# B&R Automation Studio project TD52 (part 118)

#### OUT_HACyclic.st - Cyclic code
```iecst
(*******************************************************************************
AGGR: copy OUT PVs for module HalIO (cyclic)

This code is confidential and proprietary to the INNIO Company.
It may not be used in any form, or reproduced in any manner, without the express
written permission of the INNIO Company.
Copyright, INNIO Company, 2022

Customized modifications: -
------------------------

History:
-------
V3.99	14-06-2012	Weitzer, generated FOR modular software
V4.00	14-02-2014	Weitzer, change version number
V4.00.1	29.10.2014	Weitzer, set Pact to 0 if GCB is open and -10kW < P < 10kW
V4.03	11-02-2015	Weitzer, add OUT_HA.szEng_Motorversion
		20-04-2015	Weitzer, add MORIS safety loop to MM2VIS structure
		16-09-2015	Weitzer, add MM2VIS.rP_ActUnfilt[1] for hi-res trending
		21-09-2015	Weitzer, add rI_MaxL1..3 to OUT_HA for monitoring
V4.04	17-01-2017	Denk, add IPC status OUT variables
V4.04.1	23-02-2017	Weitzer, correct current dynamic calculation
V4.05	12-09-2017	Denk, add OUT_HA.bSimWinMOD_withoutBus_Active
		27-07-2017	Messner, CAN Diagnosis Variables added
		20-12-2017	Weitzer, change bus bar voltages to standard IO format
		21-01-2018	Perktold,hardware operation mode switch added
		12.02.2018	lettenb. MM2VIS.rF_MMD_BusBar[] added
V4.05.1 14-02-2018	Weitzer, change TJ overview CAN diag. data to FAST comm.
V4.05.2 19-03-2018	Denk, WinMOD simulation ON/OFF logic added
V4.07.0	24-01-2019	Schmid, MM2VIS for MMD serial number added
V4.08	18-07-2019	Denk, IPC status logic changed because of new PPC3100 (new OUT_HA.iT_CFast2)
V4.11.0	18-03-2022	Perktold, tiTimeout von 2s auf 5s erhöht (erhöhte DGS Stabilität)
V4.12	28-10-2022	Weitzer, added auto detect multiplier for bus bar and synch voltages > 30kV
V4.14	19-11-2024	Farre,	 added auto detect multiplier for grid voltage (2024-236)

Instructions for use:
--------------------
-

Outstandings:
------------
*******************************************************************************)

PROGRAM _CYCLIC

	(* Visu out *)
	FOR ucCount := 1 TO 2 DO

		(* OUT VISU *)
		MM2VIS.rI_L1[ucCount] 			:= tI_L1[ucCount].Ai; 					(* current 1 *)
		MM2VIS.rI_L2[ucCount]			:= tI_L2[ucCount].Ai; 					(* current 2 *)
		MM2VIS.rI_L3[ucCount] 			:= tI_L3[ucCount].Ai; 					(* current 3 *)
		MM2VIS.rI_Dyn[ucCount]	 		:= UINT_TO_REAL(usIDyn[ucCount])/1000; 	(* current dynamic *)
		IF Para.rI_GenNom[ucCount] <> 0 THEN
			MM2VIS.rI_Dyn[ucCount] := UINT_TO_REAL(usIDyn[ucCount])/Para.rI_GenNom[ucCount]; 	(* current dynamic *)
		END_IF;
		MM2VIS.rI_N[ucCount] 			:= INT_TO_REAL(ssIN[ucCount]); 			(* current neutral *)
		IF ssSynchAngleDeviation[ucCount] > 1800 THEN 	(* angle deviation synchronization  +180° - -180° *)
			MM2VIS.rAng_MMD_Diff[ucCount] 	:= INT_TO_REAL(ssSynchAngleDeviation[ucCount]-3600)/10;
		ELSE
			MM2VIS.rAng_MMD_Diff[ucCount] 	:= INT_TO_REAL(ssSynchAngleDeviation[ucCount])/10;
		END_IF;

		(* visualisation of synchronization mode *)
		IF bSyncSlipMode[ucCount] THEN
			MM2VIS.iIdx_MMD_SynchMode[ucCount] := 1;
		ELSIF bSyncCheckMode[ucCount] THEN
			MM2VIS.iIdx_MMD_SynchMode[ucCount] := 2;
		ELSIF bSyncDeadBusMode[ucCount] THEN
			MM2VIS.iIdx_MMD_SynchMode[ucCount] := 3;
		ELSE
			MM2VIS.iIdx_MMD_SynchMode[ucCount] := 0;
		END_IF;

		MM2VIS.rMMD_HW_Version[ucCount]	:= UINT_TO_REAL(usMMDSynchHWVariant[ucCount])/100;			(* program version MMD *)
		MM2VIS.rU_MMD_Diff[ucCount] 	:= INT_TO_REAL(ssSynchVoltDeviation[ucCount]) * rMul_MMD_U_Synch[ucCount]; 		(* votage deviation synchronization *)
		sMMD_SerialNumber				:= UDINT_TO_STRING(ulMMDSerialNumber[ucCount]);
		MM2VIS.sMMD_SerialNumber[ucCount]	:= REPLACE(	IN1:= '00000000000', 						(* SerialNumber MMD *)
														IN2:= sMMD_SerialNumber,
														L:= LEN(sMMD_SerialNumber), P:= 11 - LEN(sMMD_SerialNumber) + 1);
		iMMD_ModuleID					:= usMMDModuleID[ucCount];
		IF iMMD_ModuleID <= 9999 THEN
			sMMD_ModuleID := UINT_TO_STRING(iMMD_ModuleID);
			sMMD_ModuleID := REPLACE(IN1:= '0000', IN2:= sMMD_ModuleID, L:= LEN(sMMD_ModuleID), P:= 4 - LEN(sMMD_ModuleID) + 1);
			MM2VIS.sMMD_SerialNumber[ucCount] := REPLACE(	IN1:= MM2VIS.sMMD_SerialNumber[ucCount], 				(* ModuleID MMD *)
															IN2:= sMMD_ModuleID,
															L:= 4, P:= 1);
		ELSE
			sMMD_ModuleID := '0000';
			FOR iIdx_ModuleID := 3 TO 0 BY -1 DO
				iMMD_ModuleID_Char	:= TRUNC(UINT_TO_REAL(iMMD_ModuleID)/16**iIdx_ModuleID);
				CASE iMMD_ModuleID_Char OF
					15:		sMMD_ModuleID	:= REPLACE(IN1:= sMMD_ModuleID, IN2:= 'F', L:= 1, P:= (4 - iIdx_ModuleID));
					14:		sMMD_ModuleID	:= REPLACE(IN1:= sMMD_ModuleID, IN2:= 'E', L:= 1, P:= (4 - iIdx_ModuleID));
					13:		sMMD_ModuleID	:= REPLACE(IN1:= sMMD_ModuleID, IN2:= 'D', L:= 1, P:= (4 - iIdx_ModuleID));
					12:		sMMD_ModuleID	:= REPLACE(IN1:= sMMD_ModuleID, IN2:= 'C', L:= 1, P:= (4 - iIdx_ModuleID));
					11:		sMMD_ModuleID	:= REPLACE(IN1:= sMMD_ModuleID, IN2:= 'B', L:= 1, P:= (4 - iIdx_ModuleID));
					10:		sMMD_ModuleID	:= REPLACE(IN1:= sMMD_ModuleID, IN2:= 'A', L:= 1, P:= (4 - iIdx_ModuleID));
					ELSE	sMMD_Temp		:= INT_TO_STRING(iMMD_ModuleID_Char);
							sMMD_ModuleID	:= REPLACE(IN1:= sMMD_ModuleID, IN2:= sMMD_Temp, L:= 1, P:= (4 - iIdx_ModuleID));
				END_CASE;
				iMMD_ModuleID		:= iMMD_ModuleID MOD REAL_TO_UINT(16**iIdx_ModuleID);
			END_FOR;
			MM2VIS.sMMD_SerialNumber[ucCount] := REPLACE(IN1:= MM2VIS.sMMD_SerialNumber[ucCount], IN2:= sMMD_ModuleID, L:= 4, P:= 1);
		END_IF;

		MM2VIS.rU_Bus_L1_2[ucCount] 	:= tU_Bus_L1_2[ucCount].Ai * rMul_MMD_U_Bus[ucCount]; 		(* bus bar voltage 1 2 *)
		MM2VIS.rU_Bus_L2_3[ucCount] 	:= tU_Bus_L2_3[ucCount].Ai * rMul_MMD_U_Bus[ucCount]; 		(* bus bar voltage 2 3 *)
		MM2VIS.rU_Bus_L3_1[ucCount] 	:= tU_Bus_L3_1[ucCount].Ai * rMul_MMD_U_Bus[ucCount]; 		(* bus bar voltage 3 1 *)
		MM2VIS.rU_Bus_L1N[ucCount] 		:= tU_Bus_L1N[ucCount].Ai  * rMul_MMD_U_Bus[ucCount]; 		(* bus bar voltage 1 *)
		MM2VIS.rU_Bus_L2N[ucCount] 		:= tU_Bus_L2N[ucCount].Ai  * rMul_MMD_U_Bus[ucCount]; 		(* bus bar voltage 2 *)
		MM2VIS.rU_Bus_L3N[ucCount] 		:= tU_Bus_L3N[ucCount].Ai  * rMul_MMD_U_Bus[ucCount]; 		(* bus bar voltage 3 *)

		(* OUT HAL_IO VIS *)
		MM2VIS.rPF_Act[ucCount]			:= tPF_Act[ucCount].Ai; 									(* power factor *)
		MM2VIS.rI_Avg[ucCount] 			:= tI_Avg[ucCount].Ai;										(* current average *)
		MM2VIS.rP_Act[ucCount]			:= tP_Act[ucCount].Ai * rMul_MMD_U_Gen[ucCount]; 			(*  actual electric power [kW] *)
		MM2VIS.rP_ActUnfilt[ucCount]	:= tP_Act[ucCount].Unfilt * rMul_MMD_U_Gen[ucCount];		(*  actual unfiltered electric power [kW] *)
		(* set to 0 kW when generator switch is open *)
		IF NOT tGCB_On.Di THEN
			IF (MM2VIS.rP_Act[1] > -10) AND (MM2VIS.rP_Act[1] < 10) THEN	(* and actual power within +/- 10 kW *)
				MM2VIS.rP_Act[1]       := 0;
				MM2VIS.rP_ActUnfilt[1] := 0;
	 		END_IF;
		END_IF;

		MM2VIS.rQ_Act[ucCount]			:= tQ_Act[ucCount].Ai 		 * rMul_MMD_U_Gen[ucCount];		(* reactive power [kVar] *)
		MM2VIS.rS_Act[ucCount]			:= tS_Act[ucCount].Ai 		 * rMul_MMD_U_Gen[ucCount];		(* power apperent *)
		MM2VIS.rU_MMD_Synch1[ucCount] 	:= tU_MMD_Synch1[ucCount].Ai * rMul_MMD_U_Synch[ucCount];	(* synchronization voltage 1 *)
		MM2VIS.rU_MMD_Synch2[ucCount] 	:= tU_MMD_Synch2[ucCount].Ai * rMul_MMD_U_Synch[ucCount];	(* synchronization voltage 2 *)
		MM2VIS.rU_Avg[ucCount] 			:= tU_Avg[ucCount].Ai 		 * rMul_MMD_U_Gen[ucCount];		(* voltage average *)
		MM2VIS.rU_L1N[ucCount]			:= tU_L1N[ucCount].Ai 		 * rMul_MMD_U_Gen[ucCount];		(* voltage 1 *)
		MM2VIS.rU_L1L2[ucCount]			:= tU_L1L2[ucCount].Ai 		 * rMul_MMD_U_Gen[ucCount];		(* voltage 12 *)
		MM2VIS.rU_L2N[ucCount]			:= tU_L2N[ucCount].Ai 		 * rMul_MMD_U_Gen[ucCount];		(* voltage 2 *)
		MM2VIS.rU_L2L3[ucCount]			:= tU_L2L3[ucCount].Ai 		 * rMul_MMD_U_Gen[ucCount];		(* voltage 23 *)
		MM2VIS.rU_L3N[ucCount]			:= tU_L3N[ucCount].Ai 		 * rMul_MMD_U_Gen[ucCount];		(* voltage 3 *)
		MM2VIS.rU_L3L1[ucCount]			:= tU_L3L1[ucCount].Ai 		 * rMul_MMD_U_Gen[ucCount]; 	(* voltage 31 *)
		MM2VIS.rF_MMD[ucCount] 			:= tF_MMD[ucCount].Ai;										(* frequency multi measure device *)
		MM2VIS.rF_MMD_Synch1[ucCount] 	:= tF_MMD_Synch1[ucCount].Ai; 								(* Frequency Sync-network 1 *)
		MM2VIS.rF_MMD_Synch2[ucCount] 	:= tF_MMD_Synch2[ucCount].Ai; 								(* Frequency Sync-network 2 *)
		MM2VIS.rF_MMD_BusBar[ucCount] 	:= tF_MMD_BusBar[ucCount].Ai; 								(* frequency bus bar *)
		MM2VIS.rMMD_FW_Version[ucCount]	:= DINT_TO_REAL(tMMD_FW_Version[ucCount].Ai)/100;			(*program version MMD firmware*)

		(* feedback synch DO *)
		TOF_SyImp[ucCount](IN := bMMD_SynchDO[ucCount],PT := T#2s);
		MM2VIS.bMMD_SynchDO[ucCount] := TOF_SyImp[ucCount].Q;

		(* U diff bar graphs MAX value (limit times 2) *)
		MM2VIS.rUDiffMaxScale[ucCount] := Para.rU_DiffMax[ucCount] * Para.rU_SyncNom[ucCount] * 2;

		(* f diff bar graphs MIN and MAX value (limit times 2) *)
		MM2VIS.rF_DiffMaxScale[ucCount] := Para.rF_DiffMax[ucCount] * 2;
		MM2VIS.rF_DiffMinScale[ucCount] := Para.rF_DiffMin[ucCount] * 2;

		(* copy maximum current values to out structure *)
		OUT_HA.rI_MaxL1[ucCount] := MM2VIS.rI_MaxL1[ucCount];
		OUT_HA.rI_MaxL2[ucCount] := MM2VIS.rI_MaxL2[ucCount];
		OUT_HA.rI_MaxL3[ucCount] := MM2VIS.rI_MaxL3[ucCount];

	END_FOR;

	(* Status MORIS safety loop for visualization *)
	MM2VIS.bMO_SaftyLoop := tMO_SaftyLoop.Di;

	(* gasmixer stepper card B&R X20 SM1426 *)
	OUT_HA.iGM1_MStepActPos; 	(*gasmixer 1 - Actual position from SM1426-Module [Microsteps]*)	(*OldName: slGM1_MStepActPos_TC1; Cycle: 5;*)
	OUT_HA.iGM1_Status;			(*gasmixer 1 - Status Word from SM1426-Module*)						(*OldName: usGM1_Status_TC1; Cycle: 5;*)
	OUT_HA.iGM2_MStepActPos;	(*gasmixer 2 - Actual position from SM1426-Module [Microsteps]*)	(*OldName: slGM2_MStepActPos_TC1; Cycle: 5;*)
	OUT_HA.iGM2_Status;			(*gasmixer 2 - Status Word from SM1426-Module*)						(*OldName: usGM2_Status_TC1; Cycle: 5;*)

	(* Copy motor version string to out structure *)
	OUT_HA.szEng_Motorversion := Para.szEng_Motorversion;

	(* Copy order ID string to out structure *)
	OUT_HA.szOrderID := Para.szOrderID;

	(* Copy order ID string to out structure *)
	OUT_HA.iEngID := VIS2MM.iEngID;

	(* IPC status *)

	OUT_HA.iSerialNumber_CPU;	(*Serial number CPU*)
	OUT_HA.iModulID_CPU;		(*Modul ID CPU*)
	OUT_HA.iPowerOnCycles;		(*Power On cycles CPU*)
	OUT_HA.iOperatingHours_CPU; (*Operating hours CPU*)
	OUT_HA.iBatterieStatus; 	(*Batterie Status IPC*)
	OUT_HA.iT_CPU; 				(*Temperature CPU*)
	OUT_HA.iT_CPU_PLC; 			(*Temperature PLC X20CP368xX CPU*)
	OUT_HA.iT_Board; 			(*Temperature Board*)
	OUT_HA.iT_Chipset;			(*Temperature Chipset*)
	OUT_HA.iT_PS; 				(*Temperature IPC board power supply*)
	OUT_HA.iT_CFast; 			(*Temperature IPC CFast*)
	OUT_HA.iT_CFast2; 			(*Temperature IPC CFast2*)

	(* WinMOD simulation for IPC status *)
	IF OUT_HA.bSimWinMOD_Active THEN
		OUT_HA.iBatterieStatus := TRUE;
	END_IF;

	(* WinMOD simulation with/without bus hardware *)
	OUT_HA.bSimWinMOD_withoutBus_Active; 	(* TRUE = without bus hardware *)

	(* WinMOD simulation ON/OFF *)
	xTON_WatchdogSIM2AR0(IN:= NOT bWatchdogSIM2AR, PT:= tiTimeout);
	xTON_WatchdogSIM2AR1(IN:= bWatchdogSIM2AR, PT:= tiTimeout);
	IF (xTON_WatchdogSIM2AR0.Q OR xTON_WatchdogSIM2AR1.Q) THEN
		OUT_HA.bSimWinMOD_Active := FALSE;
	ELSE
		OUT_HA.bSimWinMOD_Active := TRUE;
	END_IF;

	(* Status CAN BUS for Visualization *)
	MM2VIS.iCANopen_CMS_status 	:= CANopen_CMS.status;
	MM2VIS.iCANopen_CMS_info 	:= CANopen_CMS.info;
	MM2VIS.iCMSmain_Init_status	:= MAX(CMSmain_Init.status, CMSmain_Init2.status);

	(* Status CAN IC900 all Modules for Visualization *)
	MM2VIS.iIC900_AllErrEventMax 	:= IN_HA.iE_IgnStat;
	MM2VIS.iIC900_AllErrCount 		:= IN_HA.iIC900CommErrCount;
	MM2VIS.iIC900_AllErrMax 		:= ucIC900CommErrMax;
	MM2VIS.iIC900_AllPhaseCnt 		:= usIC900PhaseCnt;
	MM2VIS.iIC900_AllErrAvg			:= usIC900CommErrAvg;

	(* Status CAN Monic all Modules for Visualization *)
	MM2VIS.iMonic_AllErrEventMax 	:= IN_HA.iEMonStatus;
	MM2VIS.iMonic_AllErrCount 		:= IN_HA.iMonicCommErrCount;
	MM2VIS.iMonic_AllErrMax 		:= ucMonicCommErrMax;
	MM2VIS.iMonic_AllPhaseCnt 		:= usMonicPhaseCnt;
	MM2VIS.iMonic_AllErrAvg			:= usMonicCommErrAvg;

	(* Status CAN TecJet all Modules for Visualization - SLOW monitoring not needed *)
//	MM2VIS.iTecJet_AllErrEventMax 	:= ucTecJetCommErrEventMax;
//	MM2VIS.iTecJet_AllErrCount 		:= IN_HA.iTecJetCommErrCount;
//	MM2VIS.iTecJet_AllErrSlowMax 	:= ucTecJetCommErrSlowMax;
//	MM2VIS.iTecJet_AllSlowPhaseCnt 	:= usTecJetSlowPhaseCnt;
//	MM2VIS.iTecJet_AllErrSlowAvg	:= usTecJetCommErrSlowAvg;

	(* Status CAN TecJet individual Modules for Visualization *)
	MM2VIS.iTecJet_AllErrEventMax 	:= 0;
	MM2VIS.iTecJet_AllErrCount 		:= 0;
	MM2VIS.iTecJet_AllErrSlowMax 	:= 0;
	MM2VIS.iTecJet_AllSlowPhaseCnt 	:= 0;
	MM2VIS.iTecJet_AllErrSlowAvg	:= 0;
	FOR ucLoopCnt := 1 TO 4 DO
		MM2VIS.iTecJet_ErrEventMax[ucLoopCnt] 	:= IN_HA.tE_TEC[ucLoopCnt].Contr[0];
		MM2VIS.iTecJet_ErrMaxCur[ucLoopCnt]		:= IN_HA.iTecErrCnt[ucLoopCnt];
		MM2VIS.iTecJet_ErrMax[ucLoopCnt] 		:= usTecJetCommErrFastMax[ucLoopCnt];
		MM2VIS.iTecJet_PhaseCnt[ucLoopCnt] 		:= usTecJetFastPhaseCnt[ucLoopCnt];
		MM2VIS.iTecJet_ErrAvgCnt[ucLoopCnt] 	:= usTecJetCommErrFastAvg[ucLoopCnt];

		MM2VIS.iTecJet_AllErrEventMax 	:= MAX(MM2VIS.iTecJet_AllErrEventMax , MM2VIS.iTecJet_ErrEventMax[ucLoopCnt]);
		MM2VIS.iTecJet_AllErrCount 		:= MAX(MM2VIS.iTecJet_AllErrCount    , MM2VIS.iTecJet_ErrMaxCur[ucLoopCnt]);
		MM2VIS.iTecJet_AllErrSlowMax 	:= MAX(MM2VIS.iTecJet_AllErrSlowMax  , MM2VIS.iTecJet_ErrMax[ucLoopCnt]);
		MM2VIS.iTecJet_AllSlowPhaseCnt 	:= MAX(MM2VIS.iTecJet_AllSlowPhaseCnt, MM2VIS.iTecJet_PhaseCnt[ucLoopCnt]);
		MM2VIS.iTecJet_AllErrSlowAvg	:= MAX(MM2VIS.iTecJet_AllErrSlowAvg  , MM2VIS.iTecJet_ErrAvgCnt[ucLoopCnt]);
	END_FOR;

	(* Status CAN KLS98 all Modules for Visualization *)
	MM2VIS.iKLS98_AllErrEventMax 	:= ucKLS98CommErrEventMax;
	MM2VIS.iKLS98_AllErrMaxCur 		:= ucKLS98CommErrMaxCur;
	MM2VIS.iKLS98_AllErrMax 		:= ucKLS98CommErrMaxAll;
	MM2VIS.iKLS98_AllPhaseCntMax 	:= usKLS98PhaseCntMax;
	MM2VIS.iKLS98_AllErrAvgMax		:= usKLS98CommErrAvgMax;

	(* Status CAN KLS98 individual Modules for Visualization *)
	FOR ucLoopCnt := 1 TO xEngType.NumberOfCylinder DO
		MM2VIS.iKLS98_ErrEventMax[ucLoopCnt] 	:= IN_HA.tE_KLS[ucLoopCnt].conf[99];
		MM2VIS.iKLS98_ErrMaxCur[ucLoopCnt]		:= IN_HA.iKLS98CommErrCount[ucLoopCnt];
		MM2VIS.iKLS98_ErrMax[ucLoopCnt] 		:= ucKLS98CommErrMax[ucLoopCnt];
		MM2VIS.iKLS98_PhaseCnt[ucLoopCnt] 		:= usKLS98PhaseCnt[ucLoopCnt];
		MM2VIS.iKLS98_ErrAvgCnt[ucLoopCnt] 		:= usKLS98CommErrAvg[ucLoopCnt];
	END_FOR;

	(* Status CAN SAFI all Modules for Visualization *)
	MM2VIS.iSAFI_AllErrEventMax := ucSAFICommErrEventMax;
	MM2VIS.iSAFI_AllErrMaxCur 	:= usSAFICommErrMaxCur;
	MM2VIS.iSAFI_AllErrMax		:= usSAFICommErrMaxAll;
	MM2VIS.iSAFI_AllPhaseCntMax	:= usSAFIPhaseCntMax;
	MM2VIS.iSAFI_AllErrAvgMax	:= usSAFICommErrAvgMaxCnt;

	(* Status CAN SAFI individual Modules for Visualization *)
	FOR ucLoopCnt := 1 TO xEngType.NumberOfCylinder/2 DO
		MM2VIS.iSAFI_ErrEventMax[ucLoopCnt] := IN_HA.tE_SAFI[ucLoopCnt].sdata[1];
		MM2VIS.iSAFI_ErrMaxCur[ucLoopCnt]	:= IN_HA.iCnt_SA_ComErr[ucLoopCnt] / 100;
		MM2VIS.iSAFI_ErrMax[ucLoopCnt] 		:= usSAFICommErrMax[ucLoopCnt];
		MM2VIS.iSAFI_PhaseCnt[ucLoopCnt] 	:= usSAFIPhaseCnt[ucLoopCnt];
		MM2VIS.iSAFI_ErrAvgCnt[ucLoopCnt] 	:= usSAFICommErrAvgCnt[ucLoopCnt];
	END_FOR;

	(* H A R D W A R E   S W I T C H E S *)
	(* GoodQual for HMI *)
	OUT_HA.tHW_Switches.bGoodQual	:=  tDI_OMS_Man.GoodQual AND tDI_OMS_Auto.GoodQual AND tDI_RMS_On.GoodQual AND tDI_RMS_Remote.GoodQual AND tDI_SyOMS_Man.GoodQual AND tDI_SyOMS_Auto.GoodQual;
	(* Hardware operation mode switch *)
	xTON_OMS.IN := NOT tDI_OMS_Man.Di AND NOT tDI_OMS_Auto.Di;
	xTON_OMS();
	IF NOT tDI_OMS_Man.Di AND NOT tDI_OMS_Auto.Di AND xTON_OMS.Q THEN
		OUT_HA.tHW_Switches.iIdx_OMS_Hw 	:= 0;
	ELSIF tDI_OMS_Man.Di AND NOT tDI_OMS_Auto.Di THEN
		OUT_HA.tHW_Switches.iIdx_OMS_Hw 	:= 1;
	ELSIF NOT tDI_OMS_Man.Di AND tDI_OMS_Auto.Di THEN
		OUT_HA.tHW_Switches.iIdx_OMS_Hw 	:= 2;
	END_IF;

	(* Hardware request mode switch *)
	xTON_RMS.IN := NOT tDI_RMS_On.Di AND NOT tDI_RMS_Remote.Di;
	xTON_RMS();
	IF NOT tDI_RMS_On.Di AND NOT tDI_RMS_Remote.Di AND xTON_RMS.Q THEN
		OUT_HA.tHW_Switches.iIdx_RMS_Hw 	:= 0;
	ELSIF tDI_RMS_On.Di AND NOT tDI_RMS_Remote.Di THEN
		OUT_HA.tHW_Switches.iIdx_RMS_Hw 	:= 1;
	ELSIF NOT tDI_RMS_On.Di AND tDI_RMS_Remote.Di THEN
		OUT_HA.tHW_Switches.iIdx_RMS_Hw 	:= 2;
	END_IF;

	(* Hardware synchronisation operation mode switch *)
	xTON_SyOMS.IN := NOT tDI_SyOMS_Man.Di AND NOT tDI_SyOMS_Auto.Di;
	xTON_SyOMS();
	IF NOT tDI_SyOMS_Man.Di AND NOT tDI_SyOMS_Auto.Di AND xTON_SyOMS.Q THEN
		OUT_HA.tHW_Switches.iIdx_SyOMS_Hw 	:= 0;
	ELSIF tDI_SyOMS_Man.Di AND NOT tDI_SyOMS_Auto.Di THEN
		OUT_HA.tHW_Switches.iIdx_SyOMS_Hw 	:= 1;
	ELSIF NOT tDI_SyOMS_Man.Di AND tDI_SyOMS_Auto.Di THEN
		OUT_HA.tHW_Switches.iIdx_SyOMS_Hw 	:= 2;
	END_IF;

	(* MMU Information for custom module (bus applications) *)
	OUT_HA.rI_Dyn 				:=	MM2VIS.rI_Dyn;
	OUT_HA.rI_GenUnbalanced 	:=	MM2VIS.rI_GenUnbalanced;
	OUT_HA.rU_MMD_Diff 			:=	MM2VIS.rU_MMD_Diff;
	OUT_HA.iIdx_MMD_SynchMode 	:=	MM2VIS.iIdx_MMD_SynchMode;

END_PROGRAM
```

#### OUT_HAInit.st - Init code
```iecst
(*******************************************************************************
AGGR: copy OUT PVs for module HalIO (init)

This code is confidential and proprietary to the INNIO Company.
It may not be used in any form, or reproduced in any manner, without the express
written permission of the INNIO Company.
Copyright, INNIO Company, 2019

Customized modifications: -
------------------------

History:
-------
V3.99	06-03-2013	Weitzer, generated FOR modular software
V4.00	14-02-2014	Weitzer, change version number
V4.05	21-01-2018	Perktold,hardware operation mode switch added
V4.07	15-05-2019	Zengerer Init call for detection of missing tHA2GR items in init

Instructions for use:
--------------------
-

Outstandings:
------------
*******************************************************************************)

PROGRAM _INIT

	(* call to get a addresses for the HalIO Fub of OUT HAL_IO VIS variables *)

	PF_Act; 			(* power factor *)
	I_Avg;				(* current average *)
	P_Act; 				(*  actual electric power [kW] *)
	Q_Act; 				(* reactive power [kVar] *)
	S_Act; 				(* power apperent *)
	U_MMD_Synch1; 		(* synchronization voltage 1 *)
	U_MMD_Synch2; 		(* synchronization voltage 2 *)
	U_Avg; 				(* voltage average *)
	U_L1N; 				(* voltage 1 *)
	U_L1L2;				(* voltage 12 *)
	U_L2N; 				(* voltage 2 *)
	U_L2L3; 			(* voltage 23 *)
	U_L3N; 				(* voltage 3 *)
	U_L3L1;				(* voltage 31 *)
	F_MMD;				(* frequency multi measure device *)
	F_MMD_Synch1; 		(* Frequency Sync-network 1 *)
	F_MMD_Synch2; 		(* Frequency Sync-network 2 *)
	MMD_FW_Version;		(*program version MMD firmware*)

	xTON_OMS.PT		:= T#1s; 	(* Delaytime for changing position of HW-switch *)
	xTON_RMS.PT 	:= T#1s;	(* Delaytime for changing position of HW-switch *)
	xTON_SyOMS.PT 	:= T#1s;	(* Delaytime for changing position of HW-switch *)

	(*Init call for detection of missing tHA2GR items *)
	tHA2GR.bCheck_HA2GR ;
	tHA2GR.tU_Droop.GoodQual ;

	tHA2CU.tSet_U_Droop_COn.GoodQual ;

END_PROGRAM
```

#### OUT_HA.var - Local variables
```iecst
(********************************************************************
 * COPYRIGHT -- INNIO Company
 ********************************************************************
 * Program: IN_HA
 * File: IN_HA.var
 * Author: weitzert
 * Created: June 14, 2012
 ********************************************************************
 * Local variables of program IN_HA
 ********************************************************************)
VAR
	ucCount : USINT;
	TOF_SyImp : ARRAY[0..2] OF TOF;
	xTON_OMS : TON;
	xTON_RMS : TON;
	xTON_SyOMS : TON;
	tiTimeout : TIME := T#5s;
	xTON_WatchdogSIM2AR0 : TON;
	xTON_WatchdogSIM2AR1 : TON;
	sMMD_SerialNumber : STRING[11];
	iMMD_ModuleID : UINT;
	iMMD_ModuleID_Char : INT;
	iIdx_ModuleID : INT;
	sMMD_ModuleID : STRING[4];
	sMMD_Temp : STRING[1];
END_VAR
```

### Program Logical/HalIO/MsgHA (IEC, version 4.11.0) - + HalIO Messages

- MsgHACyclic.st (not readable text: treated as protected, skipped)

- MsgHAInit.st (not readable text: treated as protected, skipped)

#### MsgHA.var
```iecst
VAR
	iCount : USINT := 0;
	iAdrAmmBase2MM : UDINT;
	iAdrMM2AmmBase : UDINT;
	xMsg3311 : Msg;
	xMsg2399 : Msg;
	xMsg2400 : Msg;
	xMsg9400 : Msg;
	xMsg9386 : Msg; (*Plant Communication configuration failed*)
	xMsg9384 : Msg; (*Plant Communication Interrupted*)
	xMsg9391 : Msg; (*Plant Communication force active*)
END_VAR
```

### Program Logical/HalIO/ParHA (IEC, version 4.07.0) - + HalIO Parameter

- perm_par.st (not readable text: treated as protected, skipped)

#### perm_par.var
```iecst
VAR
	tParaIntern : ParaHandler_typ; (*Connector type to perm_par*)
	tMM2ParaBase_ReadBack : MM2ParaBase_type; (*INTERNAL! V4.06 new readback structure for information from previous tasks*)
	bWriteDataObj : BOOL; (* TRUE=write data object module *)
	bDataObjLenErr : BOOL; (*Error occured in permem: data module size missmatch*)
	bCreateDataObj : BOOL; (* TRUE=create new data object *)
	bWriteOnce : BOOL; (* write permanent memory once *)
	DatObjCreate_01 : DatObjCreate; (* data object create *)
	DatObjInfoBak_02 : DatObjInfo; (* data object info *)
	DatObjDelete_01 : DatObjDelete; (* data object delete *)
	DatObjRead_01 : DatObjRead; (* data object read *)
	DatObjRead_02 : DatObjRead; (* manual initiated data object read *)
	DatObjWrite_01 : DatObjWrite; (* data object write *)
	DatObjDelete_02 : DatObjDelete; (* data object delete *)
	DatObjDelete_11 : DatObjDelete; (*Delete Backup File*)
	DatObjInfo_01 : DatObjInfo; (* data object info *)
	DatObjInfo_02 : DatObjInfo; (* data object info *)
	szModuleName : STRING[35]; (* module name of object *)
	szModuleNameBackup : STRING[35]; (* module name of posiibly created backup object *)
	DatObjCopy_01 : DatObjCopy;
	bCopyDataObj : BOOL;
	TON_WarnDelay : TON;
	TON_WritePMEM : TON; (* delay write permanent memory *)
	ulPMPointer : UDINT; (* adress of actual checksum value *)
	ulChecksum : UDINT; (* parameter checksum value *)
	pm_len : UDINT; (* permanent value lenght *)
	ulChecksumOld : UDINT; (* last vlaue of parameter checksum *)
	ulChkValue : UDINT; (* actual value of parameter pointer *)
	pm_id : UDINT; (* permanent value identifier *)
	pm_p : UDINT; (* permanent value pointer *)
	DatObjInfo_META : DatObjInfo;
	DatObjRead_META : DatObjRead;
	szMetaDataRaw : STRING[2000];
	szMetaData : ARRAY[0..4] OF STRING[35];
	szMetaDataVis : ARRAY[0..3] OF STRING[35];
	ssIndex : INT;
	ssCount : INT;
	ucMetaDataRaw : ARRAY[0..2000] OF USINT;
	ssCount2 : INT;
	szMetaDataFile : STRING[10];
	szText1 : STRING[20];
	pv_adr_IN_XX_tPB2MM : UDINT;
	pv_lng : UDINT;
	pv_lng_IN_XX_tPB2MM : UDINT;
	pv_lng_OUT_XX_tPB2MM : UDINT;
	szText2 : STRING[20];
	pv_adr_OUT_XX_tXX2PB : UDINT;
END_VAR
VAR CONSTANT
	ERR_NOERROR : UINT := 0;
END_VAR
VAR
	usPMWriteCnt : UINT;
	pm_Error : UDINT; (* permanent value error *) (* Deleted: pm : ParaMem_typ; permanent memory tags mathias, 22.8.11*)
	fun_Error : UDINT := 0; (*state > 0 = function error*)
	xLocalParaCheck : ParaCheckFUB; (*local function instance to check parameter values*)
	TON_ParaSetupOk : TON;
	bParaCheckSystemOk : BOOL;
	iDebug_ParaOkChecked : UDINT;
	bRestoreBackupDataObj : BOOL := FALSE;
	bRestoreDataObjContent : BOOL := FALSE;
	pm_id_backup : UDINT;
	pm_p_Backup : UDINT;
	DatObjCopy_02 : DatObjCopy;
	bDeleteBackupDataObj : BOOL := FALSE; (*Command to delete backup data module file on purpose*)
	bDebugPara : ARRAY[0..5] OF BOOL;
	ssIndex2 : INT;
	ssIndex3 : INT;
	ssIndex4 : INT;
	ssIndexVis : INT;
	szText : STRING[40];
	pv_adr_Para : UDINT;
	szParaSnippet : ARRAY[0..5] OF STRING[150];
	szParaIndex : STRING[10];
	slValue : DINT;
	iModuleDLD_ResetCount : INT;
	bDownloadDetected : BOOL;
	bFlagParaStructCopyWorking : BOOL; (*true, if cyclic para copying is active, 1 false cycle at every copy *)
	bStoreInitParaInDataObj : BOOL := FALSE;
	bTestflag : BOOL;
	bReadOutMETA_Once : BOOL;
	tParaCheck_iPvAdress : ARRAY[0..5] OF UDINT;
	tParaCheck_iPvLengt : ARRAY[0..5] OF UDINT;
	tParaCheck_rPvValue : ARRAY[0..5] OF REAL;
	tParaCheck_rRangeMIN : ARRAY[0..5] OF REAL;
	tParaCheck_rRangeMAX : ARRAY[0..5] OF REAL;
	tParaCheck_szPvName : ARRAY[0..5] OF STRING[35];
	ssFormatDetected : INT;
	szMetaDataPart : STRING[150];
	szFullTaskName : STRING[35];
	szFullMetaModuleName : STRING[35];
	debugLen : INT;
	debugSize : INT := 0;
	strcat_adr1 : UDINT;
	strcat_adr2 : UDINT;
	ssIndexTN : INT;
	bAlternate : BOOL;
	n : INT;
	iAlternateChecksum : DINT;
	iAlternateChecksumOld : DINT;
	ulDebugChkValue : ARRAY[0..999] OF UDINT;
	Adr1 : UDINT;
	Adr2 : UDINT;
	usPMWriteCntStepsize : UINT := 1; (*different step sizes to help debug*)
	usPMWriteCntXOR : UINT;
	usPMWriteCntAltSum : UINT;
	ulAdrPM : UDINT;
	usChkValuePM : USINT;
	ulAdrPara : UDINT;
	ulPara_len : UDINT;
	usChkValuePara : USINT;
	iDebugCountPMDifferences : DINT := 0;
	bEngineRunDetected : BOOL; (*detection status bit autocommand 100 /101  for engine run state*)
	ucMetaDataDebugInfoLine : ARRAY[0..24] OF STRING[80];
	ssIndexMand : INT := 0;
	szMetaDataMand : STRING[35];
	iMyErrorInfo_Autoreset : DINT; (*internal autoreset counter*)
	ssIndex_Version : INT; (*internal*)
	ssIndex_BU : INT; (*internal*)
	ssIndex_BU2 : INT; (*internal*)
END_VAR
```

### Package Logical/HalIO/CAN - CAN

### CAN_HA.var
```iecst
(********************************************************************
 * COPYRIGHT -- INNIO Company
 ********************************************************************
 * Package: HAL_IO
 * File: CAN_HA.var
 * Author: Schmid
 * Created: December 7, 2021
 ********************************************************************
 * Variables of package HAL_IO/CAN
 ********************************************************************)
VAR CONSTANT
	iMAX_NUMB_OF_CANMODS : UINT := 20; (*Max. number of CAN modules*)
	iIdxCAN_IGN : UINT := 1; (* Ignition, Tecjet *)
	iIdxCAN_NOxS_IF1 : UINT := 2; (* NOx sensor interface 1 *)
	iIdxCAN_NOxS_IF2 : UINT := 3; (* NOx sensor interface 2 *)
	iIdxCAN_NOxS_IF3 : UINT := 7; (* NOx sensor interface 3 *)
	iIdxCAN_CB : UINT := 4; (* Conrod bearing *)
	iIdxCAN_OQS : UINT := 5; (* Oil quality sensor *)
	iIdxCAN_IGN2 : UINT := 6; (*2nd Ignition CAN line*)
	sCAN_IGN2_ident : STRING[10] := 'IGN2'; (*CAN ID string Ignition 2*)
	sCAN_IGN_ident : STRING[10] := 'IGN1'; (*CAN ID string Ignition 1*)
	sCAN_NOxS_IF1_ident : STRING[10] := 'NOX1'; (*CAN ID string NOx sensor IF1*)
	sCAN_NOxS_IF2_ident : STRING[10] := 'NOX2'; (*CAN ID string NOx sensor IF2*)
	sCAN_NOxS_IF3_ident : STRING[10] := 'NOX3'; (*CAN ID string NOx sensor IF3*)
	sCAN_CB_ident : STRING[10] := 'CRB'; (*CAN ID string Conrod bearing*)
	sCAN_OQS_ident : STRING[10] := 'OQS'; (*CAN ID string oil quality sensor*)
END_VAR
VAR
	xDiagCreateInfo_CAN : DiagCreateInfo; (*Get number of configured modules*)
	xDiagGetStrInfo_CAN : DiagGetStrInfo; (*Get name of configured modules*)
	xDiagDisposeInfo_CAN : DiagDisposeInfo; (*Free ressources of AsIODiag*)
	sLabelInfo : STRING[50]; (*Includes label of configured module*)
	sAddrInfo : STRING[50]; (*Includes address of configured modul*)
	iModPos : ARRAY[0..iMAX_NUMB_OF_CANMODS] OF UDINT; (*Array includes index of used CAN IF cards*)
	iIndex : UDINT; (*Index of actual read module*)
	iIdent : UDINT; (*Ident from xDiagCreateInfo_CAN*)
	iNrEntries : UDINT; (*Number of configured modules from xDiagCreateInfo_CAN*)
	sModSlotSel : ARRAY[0..iMAX_NUMB_OF_CANMODS] OF STRING[50]; (*Slot ID of selected configured CAN modules*)
	sCANAddr : STRING[50]; (*CAN IF PLC address string*)
	iIdxCAN_IF : ARRAY[1..2] OF UINT; (*Index array to assign CAN IF card to according role*)
	iPosCAN : ARRAY[1..2] OF UINT; (*Index array to determine CAN ID string order (for X20CS2770)*)
	iIdxPosCAN : UINT; (*Running index of found CAN IF cards*)
	xTON_CANbusoff : TON; (*CAN bus off timer*)
	xTON_SysRun : TON; (*Timer starting at PLC start*)
END_VAR
```

### Program Logical/HalIO/CAN/caninitHA (IEC, version 4.14.0) - HalIO CAN communication init

#### caninitHACyclic.st
```iecst
(*******************************************************************************
AGGR: intiate CAN communication (cyclic)

This code is confidential and proprietary to the INNIO Company.
It may not be used in any form, or reproduced in any manner, without the express
written permission of the INNIO Company.
Copyright, INNIO Company, 2024

Customized modifications: -
------------------------

History:
-------
V0.1	31-08-2001	Fahringer,	generated from caninit.c V0.2
		31-08-2001	Fahringer,	last modification
V0.21	14-10-2003	Weitzer,	transfer all CAN and CMS FUBs to caninit task
V0.40	14-02-2007  Weitzer,	change to new standard IF (SL1.SS1.IF2)
								delete MMD (multimeasure device)
V0.50	07-09-2007	Weitzer		SAFI added
								main FUB´s moved to canmain program
V0.60	23-02-2010	Weitzer,	SAFI2 (prot injection) added
V3.99.0	07-05-2012	Weitzer		generated for modular software
V4.00	14-02-2014	Weitzer,	change version number
V4.10	03-11-2020	Schmid,		engine CAN node position on node P10 as option (Aggreko standard)
V4.11	07-12-2021	Schmid,		flexible CAN interface detection
		22-12-2021	Andre,		avoid potential array index overrun
V4.12	23-02-2023	Weitzer,	add IGN2 CAN interface
V4.22	18-10-2023	Perktold,	added X20CP368xX CAN interfaces
V4.13	17-10-2023	Andre,		Only perform ARwin warm start if the CAN bus off state cannot be quit
V4.14	28-10-2024	Kafka,		SAFI / KLS21 devices of bank B use 2nd card and the rest use 1st one

Instructions for use:
--------------------
-initiate the CAN-Bus communictation controller
-initiate CAN CMS manager

Outstandings:
------------
*******************************************************************************)

PROGRAM _CYCLIC

	(* Dsiplay hardware path of CAN interface _IF1 *)

	IF MM2VIS.iCAN_HW_Slot = 0 AND IN_HA.tPB2MM.bParaSetupOk THEN

		IF LEFT(sModSlotSel[iIdxCAN_IGN],3) = LEFT(MM2VIS.sCAN_HW_Slot_X20CP368xX,3) THEN
			IF xEngType.Type9 THEN	(* B&R X20CP368xX J920 *)
				MM2VIS.iCAN_HW_Slot :=	9;
				strcpy(ADR(MM2VIS.sCAN_HW_Slot_X20CP368xX_J920), ADR(sModSlotSel[iIdxCAN_IGN]));
			ELSE					(* B&R X20CP368xX *)
				MM2VIS.iCAN_HW_Slot :=	8;
				strcpy(ADR(MM2VIS.sCAN_HW_Slot_X20CP368xX), ADR(sModSlotSel[iIdxCAN_IGN]));
			END_IF;

		ELSIF LEFT(sModSlotSel[iIdxCAN_IGN],3) = LEFT(MM2VIS.sCAN_HW_Slot_IPC_3100,3) THEN
			IF xEngType.Type9 THEN	(* B&R PPC3100 J920 *)
				MM2VIS.iCAN_HW_Slot :=	7;
				strcpy(ADR(MM2VIS.sCAN_HW_Slot_IPC_3100_J920), ADR(sModSlotSel[iIdxCAN_IGN]));
			ELSE					(* B&R PPC3100 *)
				MM2VIS.iCAN_HW_Slot :=	6;
				strcpy(ADR(MM2VIS.sCAN_HW_Slot_IPC_3100), ADR(sModSlotSel[iIdxCAN_IGN]));
			END_IF;

		ELSIF	LEFT(sModSlotSel[iIdxCAN_IGN],3) = LEFT(MM2VIS.sCAN_HW_Slot_IPC,3) THEN
			IF xEngType.Type9 THEN	(* B&R PPC900 J920 *)
				MM2VIS.iCAN_HW_Slot :=	4;
				strcpy(ADR(MM2VIS.sCAN_HW_Slot_IPC_J920), ADR(sModSlotSel[iIdxCAN_IGN]));
			ELSE					(* B&R PPC900 *)
				MM2VIS.iCAN_HW_Slot :=	1;
				strcpy(ADR(MM2VIS.sCAN_HW_Slot_IPC), ADR(sModSlotSel[iIdxCAN_IGN]));
			END_IF;

		ELSIF	LEFT(sModSlotSel[iIdxCAN_IGN],3) = LEFT(MM2VIS.sCAN_HW_Slot_IPC_GE_IP,3) THEN
			IF xEngType.Type9 THEN	(* GE IPC J920 *)
				MM2VIS.iCAN_HW_Slot :=	5;
				strcpy(ADR(MM2VIS.sCAN_HW_Slot_IPC_GE_IP_J920), ADR(sModSlotSel[iIdxCAN_IGN]));
			ELSE					(* GE IPC *)
				MM2VIS.iCAN_HW_Slot :=	3;
				strcpy(ADR(MM2VIS.sCAN_HW_Slot_IPC_GE_IP), ADR(sModSlotSel[iIdxCAN_IGN]));
			END_IF;

		ELSIF	LEFT(sModSlotSel[iIdxCAN_IGN],3) = LEFT(MM2VIS.sCAN_HW_Slot_IPC_CMaU,3) THEN
			(* B&R IPC CM&U *)
			MM2VIS.iCAN_HW_Slot	:=	2;
			strcpy(ADR(MM2VIS.sCAN_HW_Slot_IPC_CMaU), ADR(sModSlotSel[iIdxCAN_IGN]));

		ELSIF LEN(sModSlotSel[iIdxCAN_IGN]) > 0 THEN
			(* default: B&R PPC3100 *)
			MM2VIS.iCAN_HW_Slot :=	6;
			strcpy(ADR(MM2VIS.sCAN_HW_Slot_IPC_3100),	ADR(sModSlotSel[iIdxCAN_IGN]));
		END_IF;

	END_IF;

	(* cyclic call of CAN devices  *)

	IF CMSinit_Init.cms_ident <> 0 THEN		(* check if CMS init was successful *)

		IF IN_HA.tICxx_CanGo.ECANDevGo <> 0 THEN
			IF CANDevGo_InBuffer[IN_HA.tICxx_CanGo.CANDevGo[1]].ECANDevGo = 0 THEN
				CANDevGo_InBuffer[IN_HA.tICxx_CanGo.CANDevGo[1]] := IN_HA.tICxx_CanGo;
			END_IF;
		END_IF;

		IF IN_HA.tMonic_CanGo.ECANDevGo <> 0 THEN
			IF CANDevGo_InBuffer[IN_HA.tMonic_CanGo.CANDevGo[1]].ECANDevGo = 0 THEN
				CANDevGo_InBuffer[IN_HA.tMonic_CanGo.CANDevGo[1]] := IN_HA.tMonic_CanGo;
			END_IF;
		END_IF;

		IF IN_HA.tSAFI_CanGo.ECANDevGo <> 0 THEN
			IF CANDevGo_InBuffer[IN_HA.tSAFI_CanGo.CANDevGo[1]].ECANDevGo = 0 THEN
				CANDevGo_InBuffer[IN_HA.tSAFI_CanGo.CANDevGo[1]] := IN_HA.tSAFI_CanGo;
			END_IF;
		END_IF;

		IF IN_HA.tKLS98_CanGo.ECANDevGo <> 0 THEN
			IF CANDevGo_InBuffer[IN_HA.tKLS98_CanGo.CANDevGo[1]].ECANDevGo = 0 THEN
				CANDevGo_InBuffer[IN_HA.tKLS98_CanGo.CANDevGo[1]] := IN_HA.tKLS98_CanGo;
			END_IF;
		END_IF;

//		Not used at the moment
//		IF IN_HA.tGasMeteringUnit_CanGo.ECANDevGo <> 0 THEN
//			CANDevGo_InBuffer[IN_HA.tGasMeteringUnit_CanGo.CANDevGo[1]] := IN_HA.tGasMeteringUnit_CanGo;
//		END_IF;

		FOR ucDevSequencer := 1 TO 32 DO

			IF CANDevGo_InBuffer[ucDevSequencer].ECANDevGo = 128 THEN
				CANDevGo_InBuffer[ucDevSequencer].ECANDevGo := 0;
				IF ucDevSequencer < 32 THEN
					ucDevSequencer := ucDevSequencer + 1;
				END_IF;
			END_IF;

			IF CANDevGo_InBuffer[ucDevSequencer].ECANDevGo = 64 THEN
				IF ECANDevGo = 0 THEN
					CANDevGo_InBuffer[ucDevSequencer].ECANDevGo := 0;
					IF ucDevSequencer < 32 THEN
						ucDevSequencer := ucDevSequencer + 1;
					END_IF;
				ELSE
					CANDevGo_InBuffer[ucDevSequencer].ECANDevGo := 128;
				END_IF;
			END_IF;

			IF CANDevGo_InBuffer[ucDevSequencer].ECANDevGo = 1 THEN
				CANDevGo[0] := CANDevGo_InBuffer[ucDevSequencer].CANDevGo[0];
				CANDevGo[1] := ucDevSequencer;
				ECANDevGo   := 1;
				(* If only one CAN bus card was detected, all devices use it *)
				IF OUT_HA.iCANIdentIGN2 = 0 THEN
					CMSmain_Init; 		(* Cyclic starting of the CAN-manager to intitiate CAN-devices *)
				(* If 2 CAN bus cards were detected AND SAFI is active AND PI AND ignition are active, SAFI / KLS21 devices of bank B use 2nd card and the rest use 1st one *)
				ELSIF Para.bSA_Active AND Para.bSA_Ign_Active AND Para.bSA_PI_Active THEN
					IF ucDevSequencer > (9 + xEngType.NumberOfCylinder / 4) AND ucDevSequencer < (10 + xEngType.NumberOfCylinder / 2) THEN
						CMSmain_Init2; 	(* Cyclic starting of the CAN-manager to intitiate CAN-devices of 2nd CAN card *)
					ELSE
						CMSmain_Init; 	(* Cyclic starting of the CAN-manager to intitiate CAN-devices *)
					END_IF;
				(* Else all SAFI / KLS21 use the 2nd CAN bus card and the rest use the 1st one *)
				ELSE
					IF ucDevSequencer > 9 AND ucDevSequencer < 22 THEN
						CMSmain_Init2; 	(* Cyclic starting of the CAN-manager to intitiate CAN-devices of 2nd CAN card *)
					ELSE
						CMSmain_Init; 	(* Cyclic starting of the CAN-manager to intitiate CAN-devices *)
					END_IF;
				END_IF;
				CANDevGo_InBuffer[ucDevSequencer].ECANDevGo := 64;
				EXIT;
			END_IF;

		END_FOR;

		(* Copy feedback info to Out structure *)
		OUT_HA.iECanDevGo := ECANDevGo;

	END_IF;

	(* Check if CAN card started without bus off issue - if so, try to quit it. If not possible, a warm start of system is executed. *)
	xTON_SysRun(IN := TRUE, PT := T#1m);
	xTON_CANbusoff(IN := ((bCANbusoff AND bQuitCANbusoff) OR (bCANbusoff2 AND bQuitCANbusoff2)), PT := T#1s);
	IF NOT xTON_SysRun.Q THEN (* Only check during the first minute after PLC start *)
		IF bCANbusoff THEN
			bQuitCANbusoff := TRUE;
		END_IF;
		IF bCANbusoff2 THEN
			bQuitCANbusoff2 := TRUE;
		END_IF;
		IF xTON_CANbusoff.Q THEN
			SYSreset(1, 1);
		END_IF;
	END_IF;

END_PROGRAM

PROGRAM _EXIT

	(* RESET CMS TABELS *)
	CMSexit_Init(enable := TRUE, cms_ident := CMSmain_Init.cms_ident);
	CMSexit_Init(enable := TRUE, cms_ident := CMSmain_Init2.cms_ident);

END_PROGRAM
```

#### caninitHAInit.st
```iecst
(*******************************************************************************
AGGR: intiate CAN communication (init)

This code is confidential and proprietary to the INNIO Company.
It may not be used in any form, or reproduced in any manner, without the express
written permission of the INNIO Company.
Copyright, INNIO Company, 2023

Customized modifications: -
------------------------

History:
-------
V0.1	31-08-2001	Fahringer,	generated from caninit.c V0.2
		31-08-2001	Fahringer,	last modification
V0.21	14-10-2003	Weitzer,	transfer all CAN and CMS FUBs to caninit task
V0.40	14-02-2007  Weitzer,	change to new standard IF (SL1.SS1.IF2)
								delete MMD (multimeasure device)
V0.50	07-09-2007	Weitzer,	SAFI added
								main FUB´s moved to canmain program
V9.99	22-10-2007	Tinello,	Anpassung Device auf SL1.SS1.IF1
								MMDSynch
V0.60	23-02-2010	Weitzer,	SAFI2 (prot injection) added
		25-06-2010	Weitzer,	activate IF787 CAN interface, if IF787 is not available
V3.99.0	07-05-2012	Weitzer,	generated for modular software
V4.00	14-02-2014	Weitzer,	change version number
V4.03	17-03-2015	Weitzer,	add CAN open fub for J920 interface card
		22-10-2015	Weitzer,	add CAN open fub for B&R IPC hardware
V4.05	27.07.2017	Messner,	CAN Diagnosis Picture added
V4.06	18.09.2018	Denk,		don't execute task if ARsim is active
V4.08	07.02.2019	Schmid,		B&R IPC PPC3100 adaptations (PLC address for CAN device changed)
V4.10	03.11.2020	Schmid,		engine CAN node position on node P10 as option (Aggreko standard)
V4.11	07.12.2021	Schmid,		flexible CAN interface detection
V4.12	24.02.2023	Weitzer,	add IGN2 CAN interface
V4.13	17.10.2023	Andre,		moved CANbusoff check in the cyclic taks
V4.14	18.06.2024	Soto,		added CAN interface for Low NOx sensor IF3 (2023-183)

Instructions for use:
--------------------
-initiate the CAN-Bus communictation controller
-initiate CAN CMS manager

Outstandings:
------------
*******************************************************************************)

PROGRAM _INIT

	(* Don't execute task if ARsim is active *)
	IF DiagCpuIsSimulated() THEN
		strcpy(ADR(MM2VIS.sCAN_HW_Slot_IPC), ADR('Simulation active'));		(* If ARsim is active, then it's shown in CAN diagnosis picture on HMI *)
		RETURN;
	END_IF;

	(*============ GATHER CAN INTERFACE INFORMATION =============*)
	(* ********************************************************* *)
	(*	reset variables											 *)
	(* ********************************************************* *)
	memset(ADR(sLabelInfo),	 	0, SIZEOF(sLabelInfo));
	memset(ADR(sModSlotSel),	0, SIZEOF(sModSlotSel));
	memset(ADR(iModPos), 		0, SIZEOF(iModPos));

	(* ********************************************************* *)
	(*	get information about configured modules				 *)
	(* ********************************************************* *)
	xDiagCreateInfo_CAN.enable		:= TRUE;
	xDiagCreateInfo_CAN.infoKind	:= asdiagCONFIGURED;
	xDiagCreateInfo_CAN();

	IF (xDiagCreateInfo_CAN.status = 0) THEN
		iIdent 		:= xDiagCreateInfo_CAN.ident;
		iNrEntries	:= xDiagCreateInfo_CAN.nrEntries;
	END_IF;

	(* ********************************************************* *)
	(*	get name and path of configured CAN modules in Physical	 *)
	(* ********************************************************* *)
	FOR iIndex := 0 TO iNrEntries - 1 DO
		xDiagGetStrInfo_CAN.enable		:= TRUE;
		xDiagGetStrInfo_CAN.ident		:= iIdent;
		xDiagGetStrInfo_CAN.index		:= iIndex;
		xDiagGetStrInfo_CAN.infoCode	:= asdiagHARDWARE_MODULE_NAME;
		xDiagGetStrInfo_CAN.pBuffer		:= ADR(sLabelInfo);
		xDiagGetStrInfo_CAN.bufferLen	:= SIZEOF(sLabelInfo) - 1;
		xDiagGetStrInfo_CAN();

		iIdxCAN_IF[1]	:=	0;
		iIdxCAN_IF[2]	:=	0;
		iPosCAN[1]		:=	0;
		iPosCAN[2]		:=	0;
		iIdxPosCAN		:=	1;

		IF (xDiagGetStrInfo_CAN.status = 0) THEN
			(* find CAN modules *)
			IF (FIND(sLabelInfo, 'X20CS1070') <> 0) OR (FIND(sLabelInfo, 'X20CS2770') <> 0) THEN
				IF	FIND(sLabelInfo, sCAN_IGN_ident) <> 0		THEN
					iModPos[iIdxCAN_IGN]		:=	iIndex;
					iIdxCAN_IF[iIdxPosCAN]		:=	iIdxCAN_IGN;
					iPosCAN[iIdxPosCAN]			:=	FIND(sLabelInfo, sCAN_IGN_ident);
					iIdxPosCAN					:=	iIdxPosCAN + 1;
				END_IF;
				IF	FIND(sLabelInfo, sCAN_NOxS_IF1_ident) <> 0	THEN
					iModPos[iIdxCAN_NOxS_IF1]	:=	iIndex;
					iIdxCAN_IF[iIdxPosCAN]		:=	iIdxCAN_NOxS_IF1;
					iPosCAN[iIdxPosCAN]			:=	FIND(sLabelInfo, sCAN_NOxS_IF1_ident);
					iIdxPosCAN					:=	iIdxPosCAN + 1;
				END_IF;
				IF	FIND(sLabelInfo, sCAN_NOxS_IF2_ident) <> 0	THEN
					iModPos[iIdxCAN_NOxS_IF2]	:=	iIndex;
					iIdxCAN_IF[iIdxPosCAN]		:=	iIdxCAN_NOxS_IF2;
					iPosCAN[iIdxPosCAN]			:=	FIND(sLabelInfo, sCAN_NOxS_IF2_ident);
					iIdxPosCAN					:=	iIdxPosCAN + 1;
				END_IF;
				IF	FIND(sLabelInfo, sCAN_NOxS_IF3_ident) <> 0	THEN
					iModPos[iIdxCAN_NOxS_IF3]	:=	iIndex;
					iIdxCAN_IF[iIdxPosCAN]		:=	iIdxCAN_NOxS_IF3;
					iPosCAN[iIdxPosCAN]			:=	FIND(sLabelInfo, sCAN_NOxS_IF3_ident);
					iIdxPosCAN					:=	iIdxPosCAN + 1;
				END_IF;
				IF	FIND(sLabelInfo, sCAN_CB_ident) <> 0		THEN
					iModPos[iIdxCAN_CB]			:=	iIndex;
					iIdxCAN_IF[iIdxPosCAN]		:=	iIdxCAN_CB;
					iPosCAN[iIdxPosCAN]			:=	FIND(sLabelInfo, sCAN_CB_ident);
					iIdxPosCAN					:=	iIdxPosCAN + 1;
				END_IF;
				IF	FIND(sLabelInfo, sCAN_OQS_ident) <> 0		THEN
					iModPos[iIdxCAN_OQS]		:=	iIndex;
					iIdxCAN_IF[iIdxPosCAN]		:=	iIdxCAN_OQS;
					iPosCAN[iIdxPosCAN]			:=	FIND(sLabelInfo, sCAN_OQS_ident);
					iIdxPosCAN					:=	iIdxPosCAN + 1;
				END_IF;
				IF	FIND(sLabelInfo, sCAN_IGN2_ident) <> 0		THEN
					iModPos[iIdxCAN_IGN2]		:=	iIndex;
					iIdxCAN_IF[iIdxPosCAN]		:=	iIdxCAN_IGN2;
					iPosCAN[iIdxPosCAN]			:=	FIND(sLabelInfo, sCAN_IGN2_ident);
					iIdxPosCAN					:=	iIdxPosCAN + 1;
				END_IF;

				IF (iPosCAN[1] > iPosCAN[2]) AND (iPosCAN[2] <> 0) THEN
					iIdxPosCAN		:=	iIdxCAN_IF[1];	// reuse iIdxPosCAN as temporary storage variable
					iIdxCAN_IF[1]	:=	iIdxCAN_IF[2];
					iIdxCAN_IF[2]	:=	iIdxPosCAN;
				END_IF;
			END_IF;
		END_IF;

		(* ********************************************************* *)
		(*	get path of CAN modules									 *)
		(* ********************************************************* *)
		IF iIdxCAN_IF[1] <> 0 THEN
			xDiagGetStrInfo_CAN.infoCode	:= asdiagPATH;
			xDiagGetStrInfo_CAN.pBuffer		:= ADR(sAddrInfo);
			xDiagGetStrInfo_CAN.bufferLen	:= SIZEOF(sAddrInfo) - 1;
			xDiagGetStrInfo_CAN();

			IF (xDiagGetStrInfo_CAN.status = 0) THEN
				sCANAddr	:=	CONCAT(sAddrInfo,'.IF1');
				memcpy(ADR(sModSlotSel[iIdxCAN_IF[1]]), ADR(sCANAddr), SIZEOF(sModSlotSel[0])-1);
			END_IF;
			IF iIdxCAN_IF[2] <> 0 THEN
				sCANAddr	:=	CONCAT(sAddrInfo,'.IF2');
				memcpy(ADR(sModSlotSel[iIdxCAN_IF[2]]), ADR(sCANAddr), SIZEOF(sModSlotSel[0])-1);
			END_IF;
		END_IF;
	END_FOR;

	(* ********************************************************* *)
	(*	free ressources of AsIODiag								 *)
	(* ********************************************************* *)
	xDiagDisposeInfo_CAN.enable := TRUE;
	xDiagDisposeInfo_CAN.ident  := iIdent;
	xDiagDisposeInfo_CAN();
	(*===========================================================*)

	(* initialize the CAN communication controller *)

	(* enable	 := 1 						enable the functionblock CANopen      *)
	(* baud_rate := 25 						set Baud_rate - 250KB/s				  *)
	(* cob_anz	 := 500 					set maximum CMS communication objects *)
	(* error_adr := ADR(error_var)			define error - PV					  *)
	(* device	 := ADR('SL1.SS1.IF1')		Description of the interface		  *)
	(* info		 := 0						info isn't in use					  *)

	CANopen_CMS.enable		:=	1;
	CANopen_CMS.baud_rate	:=	25;
	CANopen_CMS.cob_anz		:=	500;
	CANopen_CMS.error_adr	:=	ADR(CANopen_error);
	CANopen_CMS.device		:=	ADR(sModSlotSel[iIdxCAN_IGN]);
	CANopen_CMS.info		:=	0;

	(* Default Slot Configuration - CAN Modules *)
	strcpy(ADR(MM2VIS.sCAN_HW_Slot_X20CP368xX),		ADR('IF3.ST32.IF1.ST2.IF1'));		(* B&R X20CP368xX *)
	strcpy(ADR(MM2VIS.sCAN_HW_Slot_X20CP368xX_J920),ADR('IF3.ST35.IF1.ST2.IF1'));		(* B&R X20CP368xX J920 *)
	strcpy(ADR(MM2VIS.sCAN_HW_Slot_IPC_3100),		ADR('SL2.IF1.ST32.IF1.ST2.IF1'));	(* B&R PPC3100 *)
	strcpy(ADR(MM2VIS.sCAN_HW_Slot_IPC_3100_J920),	ADR('SL2.IF1.ST35.IF1.ST2.IF1'));	(* B&R PPC3100 J920 *)
	strcpy(ADR(MM2VIS.sCAN_HW_Slot_IPC), 			ADR('SS2.IF1.ST32.IF1.ST2.IF1'));	(* B&R PPC900 *)
	strcpy(ADR(MM2VIS.sCAN_HW_Slot_IPC_J920), 		ADR('SS2.IF1.ST35.IF1.ST2.IF1'));	(* B&R PPC900 J920 *)
	strcpy(ADR(MM2VIS.sCAN_HW_Slot_IPC_CMaU), 		ADR('SS1.IF1'));					(* B&R IPC CM&U *)
	strcpy(ADR(MM2VIS.sCAN_HW_Slot_IPC_GE_IP), 		ADR('IF4.ST32.IF1.ST2.IF1'));		(* GE IPC *)
	strcpy(ADR(MM2VIS.sCAN_HW_Slot_IPC_GE_IP_J920), ADR('IF4.ST35.IF1.ST2.IF1'));		(* GE IPC J920 *)

	CANopen_CMS();

	OUT_HA.iCANIdent := CANopen_CMS.us_ident;

	(* initiate CMS manager *)

	(* enable    := 1 						enable the functionblock CANopen     *)
	(* us_ident  := CANopen_01.us_ident 	application ident  (from CANopen)    *)
	(* user_type := 0						0 ... client, 1 ... server           *)
	(* queue_cnt := 0						isn´t in use 						 *)
	(* modul_name:= ADR('cmsinit'))			name of data module with CMS objects *)

	IF CANopen_CMS.status = 0 THEN		(* check if CAN open was successful *)

		(* initiate CMS manager general *)
		CMSinit_Init(enable:=1, us_ident:=CANopen_CMS.us_ident, user_type:=0, queue_cnt:=0, modul_name:=ADR('cmsinit'));
		(* initiate CMS main function for send and receive CAN messages *)
		CMSmain_Init.enable    := TRUE;
		CMSmain_Init.cms_ident := CMSinit_Init.cms_ident;
		CMSmain_Init.cms_mode  := 2;
	ELSE
		MM2VIS.iCAN_HW_Slot := 0;
	END_IF;

	(* initialize the CAN communication controller IGN2 *)

	IF iModPos[iIdxCAN_IGN2] <> 0 THEN

		(* enable	 := 1 						enable the functionblock CANopen      *)
		(* baud_rate := 25 						set Baud_rate - 250KB/s				  *)
		(* cob_anz	 := 500 					set maximum CMS communication objects *)
		(* error_adr := ADR(error_var)			define error - PV					  *)
		(* device	 := ADR('SL1.SS1.IF1')		Description of the interface		  *)
		(* info		 := 0						info isn't in use					  *)

		CANopen_CMS.enable		:=	1;
		CANopen_CMS.baud_rate	:=	25;
		CANopen_CMS.cob_anz		:=	500;
		CANopen_CMS.error_adr	:=	ADR(CANopen_error);
		CANopen_CMS.device		:=	ADR(sModSlotSel[iIdxCAN_IGN2]);
		CANopen_CMS.info		:=	0;

		CANopen_CMS();

		OUT_HA.iCANIdentIGN2 := CANopen_CMS.us_ident;

		(* initiate CMS manager IGN2 *)

		(* enable    := 1 						enable the functionblock CANopen     *)
		(* us_ident  := CANopen_01.us_ident 	application ident  (from CANopen)    *)
		(* user_type := 0						0 ... client, 1 ... server           *)
		(* queue_cnt := 0						isn´t in use 						 *)
		(* modul_name:= ADR('cmsinit'))			name of data module with CMS objects *)

		IF CANopen_CMS.status = 0 THEN		(* check if CAN open was successful *)

			(* initiate CMS manager general *)
			CMSinit_Init(enable:=1, us_ident:=CANopen_CMS.us_ident, user_type:=0, queue_cnt:=0, modul_name:=ADR('cmsinit'));
			(* initiate CMS main function for send and receive CAN messages *)
			CMSmain_Init2.enable    := TRUE;
			CMSmain_Init2.cms_ident := CMSinit_Init.cms_ident;
			CMSmain_Init2.cms_mode  := 2;
		ELSE
			MM2VIS.iCAN_HW_Slot := 0;
		END_IF;

	END_IF;

END_PROGRAM
```

### Program Logical/HalIO/CAN/cancheckHA (IEC, version 4.05.0) - HalIO CAN communication check

#### canchkSACyclic.st
```iecst
(*******************************************************************************
AGGR: check CAN communication (cyclic)

This code is confidential and proprietary to the INNIO Company.
It may not be used in any form, or reproduced in any manner, without the express
written permission of the INNIO Company.
Copyright, INNIO Company, 2019

- read lokal counter values
- save maximum counter value
- error phase detection
- minute average

Customized modifications: -
------------------------

History:
-------
V4.05.00	27.07.2017	Messner		generated for modular software

Instructions for use:
--------------------
-

Outstandings:
------------
-
*******************************************************************************)

PROGRAM _CYCLIC

	(* Engine motortype *)
	xEngType.Motortype 	:= INT_TO_UINT(Para.iEng_Motortype);
	xEngType();

	IF xEngType.NumberOfCylinder <> 0 AND NOT OUT_HA.bSimWinMOD_Active THEN

		(*=========================================================================*)
		(* Save maximum Event Value                                                *)
		(*=========================================================================*)

		(* TecJet - save maximum event value *)
		ucTecJetCommErrEventMax := 0;

		FOR ucLoopCnt := 1 TO 4 DO
			ucTecJetCommErrEventMax := MAX(ucTecJetCommErrEventMax, IN_HA.tE_TEC[ucLoopCnt].Conf[0]);
			ucTecJetCommErrEventMax := MAX(ucTecJetCommErrEventMax, IN_HA.tE_TEC[ucLoopCnt].Conf[1]);
			ucTecJetCommErrEventMax := MAX(ucTecJetCommErrEventMax, IN_HA.tE_TEC[ucLoopCnt].Conf[2]);
			ucTecJetCommErrEventMax := MAX(ucTecJetCommErrEventMax, IN_HA.tE_TEC[ucLoopCnt].Conf[3]);
			ucTecJetCommErrEventMax := MAX(ucTecJetCommErrEventMax, IN_HA.tE_TEC[ucLoopCnt].Conf[4]);
			ucTecJetCommErrEventMax := MAX(ucTecJetCommErrEventMax, IN_HA.tE_TEC[ucLoopCnt].Conf[5]);
			ucTecJetCommErrEventMax := MAX(ucTecJetCommErrEventMax, IN_HA.tE_TEC[ucLoopCnt].Conf[6]);
			ucTecJetCommErrEventMax := MAX(ucTecJetCommErrEventMax, IN_HA.tE_TEC[ucLoopCnt].Conf[7]);
			ucTecJetCommErrEventMax := MAX(ucTecJetCommErrEventMax, IN_HA.tE_TEC[ucLoopCnt].Conf[8]);
			ucTecJetCommErrEventMax := MAX(ucTecJetCommErrEventMax, IN_HA.tE_TEC[ucLoopCnt].Status[0]);
		END_FOR;

		(*------------------------------------------------------------------------*)
		(* KLS98 - save maximum event value *)
		ucKLS98CommErrEventMax := 0;

		FOR ucLoopCnt := 1 TO xEngType.NumberOfCylinder DO

			ucKLS98CommErrEventMax		:= MAX(ucKLS98CommErrEventMax, IN_HA.tE_KLS[ucLoopCnt].conf[99]*BOOL_TO_USINT(IN_HA.tE_KLS[ucLoopCnt].conf[99] = ucKLS98EventOld[ucLoopCnt]));
			ucKLS98EventOld[ucLoopCnt]	:= IN_HA.tE_KLS[ucLoopCnt].conf[99];	(* check if event is for 2 cycle times at the same value *)

			(* start counting with value 2 because of wrong counting mode in kls98 task *)
			IF IN_HA.iKLS98CommErrCount[ucLoopCnt] > 1 THEN
				ucKLS98CommErrCountDelayed[ucLoopCnt] := IN_HA.iKLS98CommErrCount[ucLoopCnt];
			ELSE
				ucKLS98CommErrCountDelayed[ucLoopCnt] := 0;
			END_IF;
		END_FOR;

		(*------------------------------------------------------------------------*)
		(* SAFI - save maximum event value *)
		ucSAFICommErrEventMax := 0;

		FOR ucLoopCnt := 1 TO xEngType.NumberOfCylinder/2 DO
			ucSAFICommErrEventMax := MAX(ucSAFICommErrEventMax, IN_HA.tE_SAFI[ucLoopCnt].sdata[1]);
		END_FOR;

		(*------------------------------------------------------------------------*)
		(* reset max value for making new current value *)
		ucKLS98CommErrMaxCur	:= 0;
		usTecJetCommErrMaxCur	:= 0;
		usSAFICommErrMaxCur		:= 0;

		(* save maximum counter value *)
		ucIC900CommErrMax := MAX(ucIC900CommErrMax, IN_HA.iIC900CommErrCount);
		ucMonicCommErrMax := MAX(ucMonicCommErrMax, IN_HA.iMonicCommErrCount);

		ucTecJetCommErrSlowMax	:= MAX(ucTecJetCommErrSlowMax, IN_HA.iTecJetCommErrCount);
		usTecJetCommErrMaxAll	:= MAX(usTecJetCommErrMaxAll , IN_HA.iTecJetCommErrCount);
		usTecJetCommErrMaxCur	:= MAX(usTecJetCommErrMaxCur , IN_HA.iTecJetCommErrCount);

		FOR ucLoopCnt := 1 TO xEngType.NumberOfCylinder DO

			(* TecJet - maximum counter value *)
			IF ucLoopCnt <= 4 THEN
				usTecJetCommErrFastMax[ucLoopCnt] := MAX(usTecJetCommErrFastMax[ucLoopCnt], IN_HA.iTecErrCntMax[ucLoopCnt]);
				usTecJetCommErrMaxAll			  := MAX(usTecJetCommErrMaxAll			  , IN_HA.iTecErrCntMax[ucLoopCnt]);
				usTecJetCommErrMaxCur			  := MAX(usTecJetCommErrMaxCur			  , IN_HA.iTecErrCnt[ucLoopCnt]);
			END_IF;

			(* KLS98 - maximum counter value *)
			ucKLS98CommErrMax[ucLoopCnt] := MAX(ucKLS98CommErrMax[ucLoopCnt], ucKLS98CommErrCountDelayed[ucLoopCnt]);
			ucKLS98CommErrMaxAll		 := MAX(ucKLS98CommErrMaxAll		, ucKLS98CommErrCountDelayed[ucLoopCnt]);
			ucKLS98CommErrMaxCur		 := MAX(ucKLS98CommErrMaxCur		, ucKLS98CommErrCountDelayed[ucLoopCnt]);

			(* SAFI - maximum counter value *)
			IF ucLoopCnt <= xEngType.NumberOfCylinder/2 THEN
				usSAFICommErrMax[ucLoopCnt]	:= MAX(usSAFICommErrMax[ucLoopCnt], UDINT_TO_UINT(IN_HA.iCnt_SA_ComErr[ucLoopCnt] / 100));
				usSAFICommErrMaxAll			:= MAX(usSAFICommErrMaxAll		  , UDINT_TO_UINT(IN_HA.iCnt_SA_ComErr[ucLoopCnt] / 100));
				usSAFICommErrMaxCur			:= MAX(usSAFICommErrMaxCur		  , UDINT_TO_UINT(IN_HA.iCnt_SA_ComErr[ucLoopCnt] / 100));
			END_IF;

		END_FOR;

		(*=========================================================================*)
		(* Error Phase Detection                                                   *)
		(*=========================================================================*)

		(* Ignition - phase detection *)
		IF IN_HA.iIC900CommErrCount > ucCanErrLevSlowHi AND NOT bIC900PhaseDetected THEN
			bIC900PhaseDetected	:= TRUE;
			usIC900PhaseCnt		:= usIC900PhaseCnt + 1;
		END_IF;

		xTON_IC900Phase.IN := IN_HA.iIC900CommErrCount < ucCanErrLevSlowLo;
		xTON_IC900Phase.PT := T#25s;
		xTON_IC900Phase();

		IF xTON_IC900Phase.Q THEN
			bIC900PhaseDetected := FALSE;
		END_IF;

		(*------------------------------------------------------------------------*)
		(* Monic - phase detection *)
		IF IN_HA.iMonicCommErrCount > ucCanErrLevSlowHi AND NOT bMonicPhaseDetected THEN
			bMonicPhaseDetected	:= TRUE;
			usMonicPhaseCnt		:= usMonicPhaseCnt + 1;
		END_IF;

		xTON_MonicPhase.IN := IN_HA.iMonicCommErrCount < ucCanErrLevSlowLo;
		xTON_MonicPhase.PT := T#25s;
		xTON_MonicPhase();

		IF xTON_MonicPhase.Q THEN
			bMonicPhaseDetected := FALSE;
		END_IF;

		(*------------------------------------------------------------------------*)
		(* Tecjet - phase detection *)
		(* Tecjet slow communication phase detection *)
		IF IN_HA.iTecJetCommErrCount > ucCanErrLevSlowHi AND NOT bTecJetSlowPhaseDetected THEN
			bTecJetSlowPhaseDetected := TRUE;
			usTecJetSlowPhaseCnt	 := usTecJetSlowPhaseCnt + 1;
		END_IF;

		xTON_TecJetSlowPhase.IN := IN_HA.iTecJetCommErrCount < ucCanErrLevSlowLo;
		xTON_TecJetSlowPhase.PT := T#25s;
		xTON_TecJetSlowPhase();

		IF xTON_TecJetSlowPhase.Q THEN
			bTecJetSlowPhaseDetected := FALSE;
		END_IF;

		(* Tecjet fast communication phase detection *)
		FOR ucLoopCnt := 1 TO 4 DO

			IF IN_HA.iTecErrCnt[ucLoopCnt] > ucCanErrLevFastHi AND NOT bTecJetFastPhaseDetected[ucLoopCnt] THEN
				bTecJetFastPhaseDetected[ucLoopCnt]	:= TRUE;
				usTecJetFastPhaseCnt[ucLoopCnt]		:= usTecJetFastPhaseCnt[ucLoopCnt] + 1;
			END_IF;

			xTON_TecJetFastPhase[ucLoopCnt].IN := IN_HA.iTecErrCnt[ucLoopCnt] < ucCanErrLevFastLo;
			xTON_TecJetFastPhase[ucLoopCnt].PT := T#25s;
			xTON_TecJetFastPhase[ucLoopCnt]();

			IF xTON_TecJetFastPhase[ucLoopCnt].Q THEN
				bTecJetFastPhaseDetected[ucLoopCnt] := FALSE;
			END_IF;

			usTecJetFastPhaseCntMax := MAX(usTecJetFastPhaseCntMax, usTecJetFastPhaseCnt[ucLoopCnt]);

		END_FOR;

		(* Tecjet phase detection maximum *)
		usTecJetPhaseCntMax := MAX(usTecJetFastPhaseCntMax, usTecJetSlowPhaseCnt);

		(*------------------------------------------------------------------------*)
		(* KLS-98 - phase detection *)
		FOR ucLoopCnt := 1 TO xEngType.NumberOfCylinder DO

			IF ucKLS98CommErrCountDelayed[ucLoopCnt] > ucCanErrLevSlowHi AND NOT bKLS98PhaseDetected[ucLoopCnt] THEN
				bKLS98PhaseDetected[ucLoopCnt]	:= TRUE;
				usKLS98PhaseCnt[ucLoopCnt]		:= usKLS98PhaseCnt[ucLoopCnt] + 1;
			END_IF;

			xTON_KLS98Phase[ucLoopCnt].IN := ucKLS98CommErrCountDelayed[ucLoopCnt] < ucCanErrLevSlowLo;
			xTON_KLS98Phase[ucLoopCnt].PT := T#25s;
			xTON_KLS98Phase[ucLoopCnt]();

			IF xTON_KLS98Phase[ucLoopCnt].Q THEN
				bKLS98PhaseDetected[ucLoopCnt] := FALSE;
			END_IF;

			usKLS98PhaseCntMax := MAX(usKLS98PhaseCntMax, usKLS98PhaseCnt[ucLoopCnt]);

		END_FOR;

		(*------------------------------------------------------------------------*)
		(* SAFI - phase detection *)
		FOR ucLoopCnt := 1 TO xEngType.NumberOfCylinder / 2 DO

			IF DINT_TO_UINT(IN_HA.iCnt_SA_ComErr[ucLoopCnt] / 100) > ucCanErrLevSlowHi AND NOT bSAFIPhaseDetected[ucLoopCnt] THEN
				bSAFIPhaseDetected[ucLoopCnt]	:= TRUE;
				usSAFIPhaseCnt[ucLoopCnt]		:= usSAFIPhaseCnt[ucLoopCnt] + 1;
			END_IF;

			xTON_SAFIPhase[ucLoopCnt].IN := DINT_TO_UINT(IN_HA.iCnt_SA_ComErr[ucLoopCnt] / 100) < ucCanErrLevSlowLo;
			xTON_SAFIPhase[ucLoopCnt].PT := T#25s;
			xTON_SAFIPhase[ucLoopCnt]();

			IF xTON_SAFIPhase[ucLoopCnt].Q THEN
				bSAFIPhaseDetected[ucLoopCnt] := FALSE;
			END_IF;

			usSAFIPhaseCntMax := MAX(usSAFIPhaseCntMax, usSAFIPhaseCnt[ucLoopCnt]);

		END_FOR

		(*=========================================================================*)
		(* Hour Average of Error Counter                                           *)
		(*=========================================================================*)

		(* IC900 - counter increase *)
		(* count changings of counter pv´s *)
		IF ucIC900CommErrCount_Old	<> IN_HA.iIC900CommErrCount THEN
			usIC900CommErrAvgCnt	:= usIC900CommErrAvgCnt + BOOL_TO_USINT(IN_HA.iIC900CommErrCount <> 0);
			ucIC900CommErrCount_Old	:= IN_HA.iIC900CommErrCount;
		END_IF;

		(* Monic - counter increase *)
		IF ucMonicCommErrCount_Old	<> IN_HA.iMonicCommErrCount THEN
			usMonicCommErrAvgCnt 	:= usMonicCommErrAvgCnt + BOOL_TO_USINT(IN_HA.iMonicCommErrCount <> 0);
			ucMonicCommErrCount_Old := IN_HA.iMonicCommErrCount;
		END_IF;

		(* TecJet - counter increase *)
		IF ucTecJetCommErrCount_Old		<> IN_HA.iTecJetCommErrCount THEN
			usTecJetCommErrSlowAvgCnt	:= usTecJetCommErrSlowAvgCnt + BOOL_TO_USINT(IN_HA.iTecJetCommErrCount <> 0);
			usTecJetCommErrAvgMaxCnt	:= MAX(usTecJetCommErrAvgMaxCnt, usTecJetCommErrSlowAvgCnt);
			ucTecJetCommErrCount_Old	:= IN_HA.iTecJetCommErrCount;
		END_IF;

		FOR ucLoopCnt := 1 TO xEngType.NumberOfCylinder DO

			(* TecJet - counter increase *)
			IF ucLoopCnt <= 4 THEN
				IF usTecErrCnt_Old[ucLoopCnt] <> IN_HA.iTecErrCnt[ucLoopCnt] THEN
					usTecJetCommErrFastAvgCnt[ucLoopCnt] := usTecJetCommErrFastAvgCnt[ucLoopCnt] + ABS(IN_HA.iTecErrCnt[ucLoopCnt] - usTecErrCnt_Old[ucLoopCnt]);
					usTecJetCommErrAvgMaxCnt			 := MAX(usTecJetCommErrAvgMaxCnt, usTecJetCommErrFastAvgCnt[ucLoopCnt]);
					usTecErrCnt_Old[ucLoopCnt]			 := IN_HA.iTecErrCnt[ucLoopCnt];
				END_IF;
			END_IF;

			(* KLS98 - counter increase *)
			IF ucKLS98CommErrCount_Old[ucLoopCnt] <> ucKLS98CommErrCountDelayed[ucLoopCnt] THEN
				IF ucKLS98CommErrCountDelayed[ucLoopCnt] <> 0 THEN
					usKLS98CommErrAvgCnt[ucLoopCnt] := usKLS98CommErrAvgCnt[ucLoopCnt] + UINT_TO_USINT(ucKLS98CommErrCountDelayed[ucLoopCnt] - ucKLS98CommErrCount_Old[ucLoopCnt]);
				END_IF;

				usKLS98CommErrAvgMaxCnt 			:= MAX(usKLS98CommErrAvgMaxCnt, usKLS98CommErrAvgCnt[ucLoopCnt]);
				ucKLS98CommErrCount_Old[ucLoopCnt]	:= ucKLS98CommErrCountDelayed[ucLoopCnt];
			END_IF

			(* SAFI - counter increase *)
			IF ucLoopCnt <= xEngType.NumberOfCylinder/2 THEN
				IF usSAFIComErrCnt_Old[ucLoopCnt] <> DINT_TO_UINT(IN_HA.iCnt_SA_ComErr[ucLoopCnt] / 100) THEN
					usSAFICommErrAvgCnt[ucLoopCnt]	:= usSAFICommErrAvgCnt[ucLoopCnt] + BOOL_TO_USINT((IN_HA.iCnt_SA_ComErr[ucLoopCnt] / 100) <> 0);
					usSAFICommErrAvgMaxCnt			:= MAX(usSAFICommErrAvgMaxCnt, usSAFICommErrAvgCnt[ucLoopCnt]);
					usSAFIComErrCnt_Old[ucLoopCnt]	:= UDINT_TO_UINT(IN_HA.iCnt_SA_ComErr[ucLoopCnt] / 100);
				END_IF;
			END_IF;
		END_FOR;

		(*------------------------------------------------------------------------*)
		(* 1 hour max average storing *)
		usIC900CommErrAvg		:= MAX(usIC900CommErrAvg     , usIC900CommErrAvgCnt);
		usMonicCommErrAvg		:= MAX(usMonicCommErrAvg     , usMonicCommErrAvgCnt);
		usTecJetCommErrSlowAvg	:= MAX(usTecJetCommErrSlowAvg, usTecJetCommErrSlowAvgCnt);
		usTecJetCommErrAvgMax	:= MAX(usTecJetCommErrAvgMax , usTecJetCommErrAvgMaxCnt);

		FOR ucLoopCnt := 1 TO xEngType.NumberOfCylinder DO

			(* TecJet - hour average *)
			IF ucLoopCnt <= 4 THEN
				usTecJetCommErrFastAvg[ucLoopCnt] := MAX(usTecJetCommErrFastAvg[ucLoopCnt],usTecJetCommErrFastAvgCnt[ucLoopCnt]);
			END_IF;

			(* KLS98 - hour average *)
			usKLS98CommErrAvg[ucLoopCnt] := MAX(usKLS98CommErrAvg[ucLoopCnt], usKLS98CommErrAvgCnt[ucLoopCnt]);

			(* SAFI - hour average *)
			IF ucLoopCnt <= xEngType.NumberOfCylinder/2 THEN
				usSAFICommErrAvg[ucLoopCnt] := MAX(usSAFICommErrAvg[ucLoopCnt], usSAFICommErrAvgCnt[ucLoopCnt]);
			END_IF;

		END_FOR;

		usKLS98CommErrAvgMax	:= MAX(usKLS98CommErrAvgMax	, usKLS98CommErrAvgMaxCnt);
		usSAFICommErrAvgMax		:= MAX(usSAFICommErrAvgMax	, usSAFICommErrAvgMaxCnt);

		(*=========================================================================*)
		(* Reset Error Counter                                                     *)
		(*=========================================================================*)

		(* reset average counter with ervery new hour *)
		IF iCnt_OpHours_old <> IN_HA.iCnt_OpHours THEN

			usIC900CommErrAvgCnt		:= 0;
			usTecJetCommErrSlowAvgCnt	:= 0;
			usTecJetCommErrAvgMaxCnt	:= 0;

			FOR ucLoopCnt := 1 TO xEngType.NumberOfCylinder DO

				IF ucLoopCnt <= 4 THEN
					usTecJetCommErrFastAvgCnt[ucLoopCnt] := 0;
				END_IF;

				usKLS98CommErrAvgCnt[ucLoopCnt] := 0;

				IF ucLoopCnt <= xEngType.NumberOfCylinder/2 THEN
					usSAFICommErrAvgCnt[ucLoopCnt] := 0;
				END_IF;

			END_FOR;

			usKLS98CommErrAvgMaxCnt	:= 0;
			usMonicCommErrAvgCnt	:= 0;
			usSAFICommErrAvgMax		:= 0;
			iCnt_OpHours_old		:= IN_HA.iCnt_OpHours;

		END_IF;

		(*------------------------------------------------------------------------*)
		(* reset error max and phase values *)
		xTOF_CANReset.IN := VIS2MM.bCANCntReset;
		xTOF_CANReset.PT := T#1s;
		xTOF_CANReset();

		VIS2MM.bCANCntReset := FALSE;
		OUT_HA.bCANCntReset := xTOF_CANReset.Q;

		IF xTOF_CANReset.Q THEN

			(*------------------------------------------------------------------------*)
			(* reset "ERROR NUMBER" and "DEVICE GO ID" *)
			CANopen_error 					:= 0;
			IN_HA.tSAFI_CanGo.CANDevGo[1]	:= 0;

			(*------------------------------------------------------------------------*)
			(* reset maximum values *)
			ucIC900CommErrMax		:= 0;
			ucTecJetCommErrSlowMax	:= 0;
			usTecJetCommErrMax		:= 0;
			usTecJetCommErrMaxAll	:= 0;

			FOR ucLoopCnt := 1 TO xEngType.NumberOfCylinder DO

				IF ucLoopCnt <= 4 THEN
					IN_HA.iTecErrCnt[ucLoopCnt]			:= 0;		(* reset current value *)
					IN_HA.iTecErrCntMax[ucLoopCnt]		:= 0;		(* reset max value in task gas_flow *)
					usTecJetCommErrFastMax[ucLoopCnt]	:= 0;
				END_IF;

				ucKLS98CommErrMax[ucLoopCnt] := 0;

				IF ucLoopCnt <= xEngType.NumberOfCylinder/2 THEN
					usSAFICommErrMax[ucLoopCnt] := 0;
				END_IF;

			END_FOR;

			ucKLS98CommErrMaxAll	:= 0;
			ucMonicCommErrMax		:= 0;
			usSAFICommErrMaxAll		:= 0;

			(*------------------------------------------------------------------------*)
			(* reset phase counter *)
			usIC900PhaseCnt			:= 0;
			usTecJetSlowPhaseCnt	:= 0;

			FOR ucLoopCnt := 1 TO xEngType.NumberOfCylinder DO

				IF ucLoopCnt <= 4 THEN
					usTecJetFastPhaseCnt[ucLoopCnt] := 0;
				END_IF;

				usKLS98PhaseCnt[ucLoopCnt] := 0;

				IF ucLoopCnt <= xEngType.NumberOfCylinder/2 THEN
					usSAFIPhaseCnt[ucLoopCnt] := 0;
				END_IF;

			END_FOR;

			usTecJetFastPhaseCntMax	:= 0;
			usKLS98PhaseCntMax		:= 0;
			usMonicPhaseCnt			:= 0;
			usSAFIPhaseCntMax		:= 0;

			(*------------------------------------------------------------------------*)
			(* reset phase detection bits *)
			bIC900PhaseDetected		 := FALSE;
			bTecJetSlowPhaseDetected := FALSE;

			FOR ucLoopCnt := 1 TO xEngType.NumberOfCylinder DO

				IF ucLoopCnt <= 4 THEN
					bTecJetFastPhaseDetected[ucLoopCnt] := FALSE;
				END_IF;

				bKLS98PhaseDetected[ucLoopCnt] := FALSE;

				IF ucLoopCnt <= xEngType.NumberOfCylinder/2 THEN
					bSAFIPhaseDetected[ucLoopCnt] := FALSE;
				END_IF;

			END_FOR;

			bMonicPhaseDetected 	 := FALSE;

			(*------------------------------------------------------------------------*)
			(* reset average max (1h max) values *)
			usIC900CommErrAvg		:= 0;
			usTecJetCommErrSlowAvg	:= 0;
			usTecJetCommErrAvgMax	:= 0;

			FOR ucLoopCnt := 1 TO xEngType.NumberOfCylinder DO

				IF ucLoopCnt <= 4 THEN
					usTecJetCommErrFastAvg[ucLoopCnt] := 0;
				END_IF;

				usKLS98CommErrAvg[ucLoopCnt] := 0;

				IF ucLoopCnt <= xEngType.NumberOfCylinder/2 THEN
					usSAFICommErrAvg[ucLoopCnt] := 0;
				END_IF;

			END_FOR;

			usKLS98CommErrAvgMax	:= 0;
			usMonicCommErrAvg		:= 0;
			usSAFICommErrAvgMax		:= 0;

			(*------------------------------------------------------------------------*)
			(* reset average counter values *)
			usIC900CommErrAvgCnt		:= 0;
			usTecJetCommErrSlowAvgCnt	:= 0;
			usTecJetCommErrAvgMaxCnt	:= 0;

			FOR ucLoopCnt := 1 TO xEngType.NumberOfCylinder DO

				IF ucLoopCnt <= 4 THEN
					usTecJetCommErrFastAvgCnt[ucLoopCnt] := 0;
				END_IF;

				usKLS98CommErrAvgCnt[ucLoopCnt] := 0;

				IF ucLoopCnt <= xEngType.NumberOfCylinder/2 THEN
					usSAFICommErrAvgCnt[ucLoopCnt] := 0;
				END_IF;

			END_FOR;

			usKLS98CommErrAvgMaxCnt	:= 0;
			usSAFICommErrAvgMaxCnt	:= 0;
			usMonicCommErrAvgCnt	:= 0;
			iCnt_OpHours_old		:= IN_HA.iCnt_OpHours;

		END_IF;
	END_IF;

END_PROGRAM
```

#### canchkSAInit.st
```iecst
(*******************************************************************************
AGGR: check CAN communication (init)

This code is confidential and proprietary to the INNIO Company.
It may not be used in any form, or reproduced in any manner, without the express
written permission of the INNIO Company.
Copyright, INNIO Company, 2019

- get memory adresses of local counter pv´s
- error phase detection

Customized modifications: -
------------------------

History:
-------
V4.05.00	27.07.2017	Messner		generated FOR modular software

Instructions for use:
--------------------
-

Outstandings:
------------
-
*******************************************************************************)

PROGRAM _INIT

	(* error phase detection *)
	ucCanErrLevFastHi := 3;
	ucCanErrLevFastLo := 1;

	ucCanErrLevSlowHi := 5;
	ucCanErrLevSlowLo := 2;

END_PROGRAM
```

#### canchkSA.var
```iecst
VAR
	xTOF_CANReset : TOF;
	xTON_SAFIPhase : ARRAY[0..12] OF TON;
	xTON_TecJetSlowPhase : TON;
	xTON_TecJetFastPhase : ARRAY[0..4] OF TON;
	xTON_KLS98Phase : ARRAY[0..24] OF TON;
	xTON_IC900Phase : TON;
	xTON_MonicPhase : TON;
	bSAFIPhaseDetected : ARRAY[0..12] OF BOOL;
	usSAFIComErrCnt_Old : ARRAY[0..12] OF UINT; (* counter for SAFI comm. problem *)
	bTecJetSlowPhaseDetected : BOOL;
	bTecJetFastPhaseDetected : ARRAY[0..4] OF BOOL;
	usTecJetCommErrAvgMaxCnt : UINT;
	usTecErrCnt_Old : ARRAY[0..4] OF UINT;
	ucTecJetCommErrCount_Old : USINT; (* counter for KLS98 comm. problem *)
	usTecJetCommErrSlowAvgCnt : USINT;
	usTecJetCommErrFastAvgCnt : ARRAY[0..4] OF UINT;
	bKLS98PhaseDetected : ARRAY[0..24] OF BOOL;
	ucKLS98CommErrCountDelayed : ARRAY[0..24] OF USINT;
	usKLS98CommErrAvgCnt : ARRAY[0..24] OF UINT;
	usKLS98CommErrAvgMaxCnt : UINT;
	ucKLS98CommErrCount_Old : ARRAY[0..24] OF USINT;
	ucKLS98EventOld : ARRAY[0..24] OF USINT;
	bMonicPhaseDetected : BOOL;
	usMonicCommErrAvgCnt : UINT;
	ucMonicCommErrCount_Old : USINT; (* counter for Monic comm. problem *)
	bIC900PhaseDetected : BOOL;
	usIC900CommErrAvgCnt : UINT;
	ucIC900CommErrCount_Old : USINT; (* counter for KLS98 comm. problem *)
	ucCanErrLevSlowHi : USINT;
	ucCanErrLevSlowLo : USINT;
	ucCanErrLevFastHi : USINT;
	ucCanErrLevFastLo : USINT;
END_VAR
```

### Program Logical/HalIO/CAN/CAN_NOx_WG (IEC, version 4.14.0) - HalIO get CAN device ID for NOx sensor and WG actuators

#### CAN_NOx_WGInit.st - Initialization code
```iecst
(*******************************************************************************
AGGR: intiate CAN communication for NOx sensor and WG actuators (init)

This code is confidential and proprietary to the INNIO Company.
It may not be used in any form, or reproduced in any manner, without the express
written permission of the INNIO Company.
Copyright, INNIO Company, 2021

Customized modifications: -
------------------------

History:
-------
V3.99.0	07-05-2012	Weitzer,	generated FOR modular software
V4.00	14-02-2014	Weitzer,	change version number
V4.03	22-10-2015	Weitzer,	add interface for B&R IPC hardware
V4.05	02-08-2017	Tinello,	add interface for two sensors
V4.06	18.09.2018	Denk,		don't execute task if ARsim is active
V4.07	04.04.2019	Tinello,	two fixed CAN adresses for NOx
V4.08	07.02.2019	Schmid,		B&R IPC PPC3100 adaptations (PLC address for CAN device changed)
V4.09	01.12.2019	Tinello,	added variables for CANopen HMI overview
V4.10	03.11.2020	Schmid,		engine NOx CAN node position on node P21 as option
V4.11	07.12.2021	Schmid,		flexible CAN interface detection
V4.14	28.03.2024	Soto/Farre,	change task name, CAN NOx IF1 shared with Wastegate, interfaces duplicated (2023-174)
		18.06.2024	Soto,		added CAN interface for Low NOx sensor IF3 (2023-183)

*******************************************************************************)

PROGRAM _INIT

	(* Do not execute task if ARsim is active *)
	IF DiagCpuIsSimulated() THEN
		RETURN;
	END_IF;

	(* initialize the CAN communication for NOx-sensors *)
	MM2VIS.sCAN_HW_NOxS_IF1 := CONCAT(sModSlotSel[iIdxCAN_NOxS_IF1],' /EX=1');	(* Address of CAN interface 1 *)

	xCANopen_NOxS_IF1.enable	:= 1;										(* enable the functionblock CANopen *)
	xCANopen_NOxS_IF1.baud_rate := 25;										(* set baut rate - 250kB/s *)
	xCANopen_NOxS_IF1.cob_anz	:= 50;										(* set maximum communication objects *)
	xCANopen_NOxS_IF1.error_adr	:= ADR(iCANopen_NOxS_Err_IF1);				(* description of the error *)
	xCANopen_NOxS_IF1.device	:= ADR(MM2VIS.sCAN_HW_NOxS_IF1);			(* assign device at BR hardware *)
	xCANopen_NOxS_IF1.info	  	:= 0;							  	  		(* info is not in use *)
	xCANopen_NOxS_IF1;														(* execute of the CANopen *)

	IF xCANopen_NOxS_IF1.status <> 0 THEN
		strcpy(ADR(MM2VIS.sCAN_HW_NOxS_IF1), ADR('INTERFACE NOT FOUND'));	(* node not configured or no identifier label *)
	ELSE
		OUT_HA.iCAN_NOxS_IF1_us_ident	:= xCANopen_NOxS_IF1.us_ident;
	END_IF;

	(* initialize the CAN communication for NOx-sensors with different CAN devices *)
	MM2VIS.sCAN_HW_NOxS_IF2 := CONCAT(sModSlotSel[iIdxCAN_NOxS_IF2],' /EX=1');	(* Address of CAN interface 2 *)

	xCANopen_NOxS_IF2.enable	:= 1;										(* enable the functionblock CANopen *)
	xCANopen_NOxS_IF2.baud_rate := 25;										(* set baut rate - 250kB/s *)
	xCANopen_NOxS_IF2.cob_anz  	:= 50;										(* set maximum communication objects *)
	xCANopen_NOxS_IF2.error_adr := ADR(iCANopen_NOxS_Err_IF2);				(* description of the error *)
	xCANopen_NOxS_IF2.device    := ADR(MM2VIS.sCAN_HW_NOxS_IF2);			(* assign device at BR hardware *)
	xCANopen_NOxS_IF2.info	  	:= 0;							  	  		(* info is not in use *)
	xCANopen_NOxS_IF2;														(* execute of the CANopen *)

	IF xCANopen_NOxS_IF2.status <> 0 THEN
		strcpy(ADR(MM2VIS.sCAN_HW_NOxS_IF2), ADR('INTERFACE NOT FOUND'));	(* node not configured or no identifier label *)
	ELSE
		OUT_HA.iCAN_NOxS_IF2_us_ident	:= xCANopen_NOxS_IF2.us_ident;
	END_IF;

	(* initialize the CAN communication for NOx-sensors with different CAN devices *)
	MM2VIS.sCAN_HW_NOxS_IF3 := CONCAT(sModSlotSel[iIdxCAN_NOxS_IF3],' /EX=0');		(* Address of CAN interface 3 *)

	xCANopen_NOxS_IF3.enable	:= 1;										(* enable the functionblock CANopen *)
	xCANopen_NOxS_IF3.baud_rate := 50;										(* set baut rate - 500kB/s *)
	xCANopen_NOxS_IF3.cob_anz  	:= 50;										(* set maximum communication objects *)
	xCANopen_NOxS_IF3.error_adr := ADR(iCANopen_NOxS_Err_IF3);				(* description of the error *)
	xCANopen_NOxS_IF3.device    := ADR(MM2VIS.sCAN_HW_NOxS_IF3);			(* assign device at BR hardware *)
	xCANopen_NOxS_IF3.info	  	:= 0;							  	  		(* info is not in use *)
	xCANopen_NOxS_IF3;														(* execute of the CANopen *)

	IF xCANopen_NOxS_IF3.status <> 0 THEN
		strcpy(ADR(MM2VIS.sCAN_HW_NOxS_IF3), ADR('INTERFACE NOT FOUND'));	(* node not configured or no identifier label *)
	ELSE
		OUT_HA.iCAN_NOxS_IF3_us_ident	:= xCANopen_NOxS_IF3.us_ident;
	END_IF;

	MM2VIS.iCANopen_NOxS_IF1_status		:= xCANopen_NOxS_IF1.status;
	MM2VIS.iCANopen_NOxS_IF2_status		:= xCANopen_NOxS_IF2.status;
	MM2VIS.iCANopen_NOxS_IF3_status		:= xCANopen_NOxS_IF3.status;

	(* CAN Wastegate - duplicate interface from NOx shared interface IF1 *)
	OUT_HA.iCAN_WG_us_ident 	:= OUT_HA.iCAN_NOxS_IF1_us_ident; 			(* CAN WG identifier *)
	MM2VIS.sCAN_HW_WG			:= MM2VIS.sCAN_HW_NOxS_IF1;					(* BR Adress of CAN interface 1 *)
	MM2VIS.iCANopen_WG_status	:= MM2VIS.iCANopen_NOxS_IF1_status;			(* CAN WG status *)

END_PROGRAM
```

#### CAN_NOx_WG.var - Local variables
```iecst
VAR
	iCANopen_NOxS_Err_IF1 : UDINT; (* description of the interface 1 define error*) (* OldName: usCANopenUniNOx_error; Cycle:8; *)
	iCANopen_NOxS_Err_IF2 : UDINT; (* description of the interface 2 define error*) (* OldName: usCANopenUniNOx_error; Cycle:8; *)
	iCANopen_NOxS_Err_IF3 : UDINT; (* description of the interface 3 define error*) (* OldName: usCANopenUniNOx_error; Cycle:8; *)
	xCANopen_NOxS_IF1 : CANopen; (* CANopen NOx sensor interface 1*) (* OldName: CANopen_UniNOx; Cycle:8; *)
	xCANopen_NOxS_IF2 : CANopen; (* CANopen NOx sensor interface 2*) (* OldName: CANopen_UniNOx; Cycle:8; *)
	xCANopen_NOxS_IF3 : CANopen; (* CANopen NOx sensor interface 3*) (* OldName: CANopen_UniNOx; Cycle:8; *)
END_VAR
```

### Program Logical/HalIO/CAN/CAN_Conrod (IEC, version 4.11.0) - HalIO get CAN device ID for NOx sensor

#### CAN_ConrodInit.st - Initialization code
```iecst
(*******************************************************************************
AGGR: intiate CAN communication for conrod bearing system (init)

This code is confidential AND proprietary to the INNIO Company.
It may NOT be used in any form, or reproduced in any manner, without the express
written permission of the INNIO Company.
Copyright, INNIO Company, 2021

Customized modifications: -
------------------------

History:
-------
V4.03	23-02-2015	Tinello,	new
		22-10-2015	Weitzer,	add interface for B&R IPC hardware
V4.06	18.09.2018	Denk,		don't execute task if ARsim is active
V4.08	07.02.2019	Schmid,		B&R IPC PPC3100 adaptations (PLC address for CAN device changed)
V4.11	07.12.2021	Schmid,		flexible CAN interface detection

Instructions FOR use:
--------------------
-initiate the CAN-Bus communictation controller

Outstandings:
------------
*******************************************************************************)

PROGRAM _INIT

	(* Don't execute task if ARsim is active *)
	IF DiagCpuIsSimulated() THEN
		RETURN;
	END_IF;

	(* initialize the CAN communication controller *)
	xCANopen_CB.enable	 	:= TRUE;
	xCANopen_CB.baud_rate 	:= 25;								(* set baud rate - 250kB/s *)
	xCANopen_CB.cob_anz		:= 500;								(* set maximum communication objects *)
	xCANopen_CB.error_adr 	:= ADR(iCANopen_CB_Err);			(* description of the interface define error *)
	xCANopen_CB.device	 	:= ADR(sModSlotSel[iIdxCAN_CB]);	(* assign device at B&R PPC3100 hardware *)
	xCANopen_CB.info		:= 0;								(* info isn´t in use *)
	xCANopen_CB();

	IF xCANopen_CB.status = 0 THEN
		OUT_HA.iCAN_CB_us_ident := xCANopen_CB.us_ident;
	ELSE
		OUT_HA.iCAN_CB_us_ident := 0;
	END_IF;

END_PROGRAM
```

#### CAN_Conrod.var - Local variables
```iecst
VAR
	xCANopen_CB : CANopen := (0); (*FuB*)
	iCANopen_CB_Err : UDINT := 0; (*error variable for the CAN FUB*)
END_VAR
```

### Program Logical/HalIO/CAN/CAN_OQS (IEC, version 4.08.0) - HalIO get CAN device ID for OQS sensor

#### CAN_OQSInit.st - Initialization code
```iecst
(*******************************************************************************
AGGR: intiate CAN communication for oil quality sensor (init)

This code is confidential AND proprietary to the INNIO Company.
It may NOT be used in any form, or reproduced in any manner, without the express
written permission of the INNIO Company.
Copyright, INNIO Company, 2021

Customized modifications: -
------------------------

History:
-------
V4.11	05.11.2021	Schmid,		new CAN interface for oil quality sensor

Instructions FOR use:
--------------------
-initiate the CAN-Bus communictation controller

Outstandings:
------------
*******************************************************************************)

PROGRAM _INIT

	(* Don't execute task if ARsim is active *)
	IF DiagCpuIsSimulated() THEN
		RETURN;
	END_IF;

	(* initialize the CAN OQS OC communication controller *)
	xCANopen_OQS_OC.enable	 	:= TRUE;
	xCANopen_OQS_OC.baud_rate 	:= 12;								(* set baud rate - 125kB/s *)
	xCANopen_OQS_OC.cob_anz		:= 500;								(* set maximum communication objects *)
	xCANopen_OQS_OC.error_adr 	:= ADR(iCANopen_OQS_OC_Err);		(* description of the interface define error *)
	xCANopen_OQS_OC.device	 	:= ADR(sModSlotSel[iIdxCAN_OQS]);	(* assign device at B&R PPC3100 hardware *)
	xCANopen_OQS_OC.info		:= 0;								(* info isn´t in use *)
	xCANopen_OQS_OC();

	IF xCANopen_OQS_OC.status = 0 THEN
		OUT_HA.iCAN_OQS_OC_us_ident := xCANopen_OQS_OC.us_ident;
	ELSE
		OUT_HA.iCAN_OQS_OC_us_ident := 0;
	END_IF;

END_PROGRAM
```

#### CAN_OQS.var - Local variables
```iecst
VAR
	xCANopen_OQS_OC : CANopen := (0); (*FuB*)
	iCANopen_OQS_OC_Err : UDINT := 0; (*error variable for the CAN OQS OC FUB*)
END_VAR
```

### Data object Logical/HalIO/CAN/cmsinit (Simple, version 4.00.0) - HalIO CAL init

#### cmsinit.dat
```
; *******************************************************************************
; AGGR: client cmsinit (data module)
; Copyright 1998 - 2014 GE Jenbacher
;
; - init CAN CMS communication
;
; Customized modifications: -
; ------------------------
;
; History:
; -------
; V1.1	30-04-1999	Fahringer, generated
; 		30-04-1999	Fahringer, last modification
; V3.99	07-05-2012	Weitzer,   generated for modular software
; V4.00	14-02-2014	Weitzer,   change version number
;
; Instructions for use:
; --------------------
;
; Outstandings:
; ------------
;
; *******************************************************************************
;   structure of entry
;   ------------------
;   str       startstring
;   client    client CAN identifier
;   server    server CAN identifier
;   acc       access_typ (R=ReadOnly, W=WriteOnly, A=Read/Write)
;   obj       object_typ (B=Basic variable, M=Multiplexed variable,
;						  U=uncontroled event)
;   mul       multiplexer for multiplexed variable (0-127)
;   len       length (not used)
;   info      info (0=CiA/DS202-3, 1=BigEndian Motorola format)
;   variable  name of variable (max.strlen=31 Byte) (global)
;   event_pv  name of event variable (max.32 Byte) (TYP=BYTE) (global)
;
; str| client | server  |acc|obj|mul|  len   |  info  |   variable   | event_pv
;-------------------------------------------------------------------------------

; Device Start-Stop
"%P",$00000000,$00000000,'W','B',000,00000000,00000000,"HalIO::CANDevGo","HalIO::ECANDevGo"
```

### Data object Logical/HalIO/IOcfg (Simple, version 4.00.0) - HalIO IO configuration

- IOcfg.dat (not shown)

### Data object Logical/HalIO/IOcfgAll (Simple, version 4.25.0) - HalIO All IO configurations

- IOcfgAll.dat (not shown)

### Data object Logical/HalIO/IOcfgAll_UR20 (Simple, version 4.25.0) - HalIO All IO configurations

- IOcfgAll_UR20.dat (not shown)

### PlantComVariables.var
```iecst
(*Diagnostics*)
VAR
	tDiagClient : DiagClient_Struct := (0); (*ANSL Client Diagnostics*)
	tDiagEngine : ARRAY[0..32] OF DiagConn_Struct := [33((0))]; (*ANSL Communication Diagnostics for Engine Communication*)
	tDiagMaster : ARRAY[0..4] OF DiagConn_Struct := [5((0))]; (*ANSL Communication Diagnostics for Master Communication*)
	iNum_InterruptedEngines : USINT := 0; (*Number of interrupted communications to engines*)
	iNum_InterruptedMasters : USINT := 0; (*Number of interrupted communications to masters*)
END_VAR
(*General Communication Variables*)
VAR
	bRedundantMasterEnabled : BOOL := FALSE; (*Enable if master control is redundant*)
	bEng2EngComEnabled : BOOL := FALSE; (*Enabled if valid parameters for Engine Number Min and Max are supplied, disabled for min and max = 0*)
	bEng2MasComEnabled : BOOL := FALSE; (*Enabled if valid parameters for Master Number Min and Max are supplied, disabled for min and max = 0*)
	iEngNumMin : USINT := 0; (*First Engine Number  in in the communication*)
	iEngNumMax : USINT := 0; (*Last Engine Number in the communication*)
	iMasNumMax : USINT := 0; (*Last Master Number in the communication*)
	iMasNumMin : USINT := 0; (*First Master Number in the communication*)
	iSelectedMaster : USINT := 1; (*Master that is controling this engine. Default master 1*)
END_VAR
(*ANSL Communication Output/Input Data Variables*)
VAR
	tPlantCom_M2E_In_10ms : ARRAY[0..4] OF tData_M2E_10ms_Struct := [5((0))]; (*Fast Inputs (Master -> Engine)*)
	tPlantCom_E2M_Out_10ms : ARRAY[0..4] OF tData_E2M_10ms_Struct := [5((0))]; (*Fast Outputs (Engine -> Master)*)
	tPlantCom_E2E_In_10ms : ARRAY[0..32] OF tData_E2E_10ms_Struct := [33((0))]; (*Fast Inputs (Engine -> Engine)*)
	tPlantCom_E2E_Out_10ms : tData_E2E_10ms_Struct := (0); (*Fast Outputs (Engine -> Engine)*)
	tPlantCom_M2E_In_100ms : ARRAY[0..4] OF tData_M2E_100ms_Struct := [5((0))]; (*Slow Inputs (Master -> Engine)*)
	tPlantCom_E2M_Out_100ms : ARRAY[0..4] OF tData_E2M_100ms_Struct := [5((0))]; (*Slow Outputs (Engine -> Master)*)
	tPlantCom_E2E_In_100ms : ARRAY[0..32] OF tData_E2E_100ms_Struct := [33((0))]; (*Slow Inputs (Engine -> Engine)*)
	tPlantCom_E2E_Out_100ms : tData_E2E_100ms_Struct := (0); (*Slow Outputs (Engine -> Engine)*)
END_VAR
(*Plant Communication Data Variables*)
VAR
	tPlantCom_E2E_Out_Hmi : tHmiDiagnosticData := (0); (*HMI Data Outputs (Engine -> Engine)*)
	tPlantCom_E2E_In_Hmi : ARRAY[0..32] OF tHmiDiagnosticData := [33((0))]; (*HMI Data Inputs (Engine -> Engine)*)
	tPlantCom_E2M_Out_Hmi : ARRAY[0..4] OF tHmiDiagnosticData := [5((0))]; (*HMI Data Outputs (Engine -> Master)*)
	tPlantCom_M2E_In_Hmi : ARRAY[0..4] OF tHmiDiagnosticData := [5((0))]; (*HMI Data Inputs (Master  -> Engine)*)
	tPlantCom_E2E_Out_Bus : tPlantComData_EngEng_Struct := (0); (*Bus Data Outputs (Engine -> Engine)*)
	tPlantCom_E2E_In_Bus : ARRAY[0..32] OF tPlantComData_EngEng_Struct := [33((0))]; (*Bus Data Inputs (Engine -> Engine)*)
	tPlantCom_E2M_Out_Bus : ARRAY[0..4] OF tPlantComData_EngEng_Struct := [5((0))]; (*Bus Data Outputs (Engine -> Master)*)
	tPlantCom_M2E_In_Bus : ARRAY[0..4] OF tPlantComData_EngMas_Struct := [5((0))]; (*Bus Data Inputs (Master  -> Engine)*)
	tPlantCom_E2E_Out_Plc : tPlantComData_EngEng_Struct := (0); (*Plc Data Outputs (Engine -> Engine)*)
	tPlantCom_E2E_In_Plc : ARRAY[0..32] OF tPlantComData_EngEng_Struct := [33((0))]; (*Plc Data Inputs (Engine -> Engine)*)
	tPlantCom_E2M_Out_Plc : ARRAY[0..4] OF tPlantComData_EngEng_Struct := [5((0))]; (*Plc Data Outputs (Engine -> Master)*)
	tPlantCom_M2E_In_Plc : ARRAY[0..4] OF tPlantComData_EngMas_Struct := [5((0))]; (*Plc Data Inputs (Master  -> Engine)*)
	tPlantCom_M2E_In_Active : ARRAY[0..4] OF tPlantComActive_EngMas_Struct := [5((0))];
	tPlantCom_E2E_In_Active : ARRAY[0..32] OF tPlantComActive_EngEng_Struct := [33((0))];
END_VAR
(*Plant Communication Array Size Constants*)
VAR CONSTANT
	iAnaArrayMaxAll : USINT := iAnaArrayMax10ms+iAnaArrayMax100ms+1; (*Number of Analog Signals (Fast + Slow)*)
	iDigArrayMaxAll : USINT := iDigArrayMax10ms+iDigArrayMax100ms+1; (*Number of Digital Signals (Fast + Slow)*)
	iAnaArrayMax10ms : USINT := 15; (*Number of Fast Analog Signals*)
	iDigArrayMax10ms : USINT := 31; (*Number of Fast Digital Signals*)
	iAnaArrayMax100ms : USINT := 31; (*Number of Slow Analog Signals*)
	iDigArrayMax100ms : USINT := 63; (*Number of Slow Digital Signals*)
END_VAR
```

### PlantComTypes.typ
```iecst
(*PlantCommunication Diagnostic Structures*)

TYPE
	DiagClient_Struct : 	STRUCT  (*ANSL Client Diagnostics Data*)
		Conn : UDINT;
		ConnErr : UDINT;
		TimeStamp : AsANSLTimeStampType;
	END_STRUCT;
	DiagConn_Struct : 	STRUCT  (*ANSL Connection Diagnostics Data*)
		Err : UDINT;
		PvWrite : UDINT;
		PvWriteErr : UDINT;
		PvReadErr : UDINT;
		RedConnActIpAddr : UDINT;
		RedConnAct : UDINT;
		RedConnState : UDINT;
	END_STRUCT;
END_TYPE

(*PlantCommunication Data Structures*)

TYPE
	tData_E2M_100ms_Struct : 	STRUCT  (*Slow Data sent from Engine to Master*)
		digitalSignals : ARRAY[0..iDigArrayMax100ms]OF tDigitalSignal_Struct; (*Digital Outputs with GoodQual*)
		analogSignals : ARRAY[0..iAnaArrayMax100ms]OF tAnalogSignal_Struct; (*Analog Inputs with GoodQual*)
	END_STRUCT;
	tData_M2E_100ms_Struct : 	STRUCT  (*Slow Data sent from Master to Engine*)
		digitalSignals : ARRAY[0..iDigArrayMax100ms]OF tDigitalSignal_Struct; (*Digital Inputs with GoodQual*)
		analogSignals : ARRAY[0..iAnaArrayMax100ms]OF tAnalogSignal_Struct; (*Analog Inputs with GoodQual*)
	END_STRUCT;
	tData_E2E_100ms_Struct : 	STRUCT  (*Slow Data set from Engine to Engine*)
		digitalSignals : ARRAY[0..iDigArrayMax100ms]OF tDigitalSignal_Struct; (*Digital Signals with GoodQual*)
		analogSignals : ARRAY[0..iAnaArrayMax100ms]OF tAnalogSignal_Struct; (*Analog Signals with GoodQual*)
	END_STRUCT;
	tData_E2M_10ms_Struct : 	STRUCT  (*Fast Data sent from Engine to Master*)
		digitalSignals : ARRAY[0..iDigArrayMax10ms]OF tDigitalSignal_Struct; (*Digital Outputs with GoodQual*)
		analogSignals : ARRAY[0..iAnaArrayMax10ms]OF tAnalogSignal_Struct; (*Analog Inputs with GoodQual*)
	END_STRUCT;
	tData_M2E_10ms_Struct : 	STRUCT  (*Fast Data sent from Master to Engine*)
		digitalSignals : ARRAY[0..iDigArrayMax10ms]OF tDigitalSignal_Struct; (*Digital Inputs with GoodQual*)
		analogSignals : ARRAY[0..iAnaArrayMax10ms]OF tAnalogSignal_Struct; (*Analog Inputs with GoodQual*)
	END_STRUCT;
	tData_E2E_10ms_Struct : 	STRUCT  (*Fast Data set from Engine to Engine*)
		digitalSignals : ARRAY[0..iDigArrayMax10ms]OF tDigitalSignal_Struct; (*Digital Signals with GoodQual*)
		analogSignals : ARRAY[0..iAnaArrayMax10ms]OF tAnalogSignal_Struct; (*Analog Signals with GoodQual*)
	END_STRUCT;
	tHmiDiagnosticData : 	STRUCT  (*HMI Diagnostics Data*)
		bDigForceActive : ARRAY[0..iDigArrayMaxAll]OF BOOL;
		bAnaForceActive : ARRAY[0..iAnaArrayMaxAll]OF BOOL;
		rForceValue : ARRAY[0..iAnaArrayMaxAll]OF REAL;
		bForceValue : ARRAY[0..iDigArrayMaxAll]OF BOOL;
		iCommentNr : USINT;
		iNum_ForcedValues : USINT;
	END_STRUCT;
	tPlantComData_EngEng_Struct : 	STRUCT  (*Data shared between the Engines*)
		digitalSignals : ARRAY[0..iDigArrayMaxAll]OF tDigitalSignal_Struct;
		analogSignals : ARRAY[0..iAnaArrayMaxAll]OF tAnalogSignal_Struct;
	END_STRUCT;
	tPlantComData_EngMas_Struct : 	STRUCT  (*Data shared between the Master and the Engines*)
		digitalSignals : ARRAY[0..iDigArrayMaxAll]OF tDigitalSignal_Struct;
		analogSignals : ARRAY[0..iAnaArrayMaxAll]OF tAnalogSignal_Struct;
	END_STRUCT;
	tPlantComActive_EngEng_Struct : 	STRUCT
		digitalSignalActive : ARRAY[0..iDigArrayMaxAll]OF BOOL;
		analogSignalActive : ARRAY[0..iAnaArrayMaxAll]OF BOOL;
	END_STRUCT;
	tPlantComActive_EngMas_Struct : 	STRUCT
		digitalSignalActive : ARRAY[0..iDigArrayMaxAll]OF BOOL;
		analogSignalActive : ARRAY[0..iAnaArrayMaxAll]OF BOOL;
	END_STRUCT;
END_TYPE
```

### Program Logical/HalIO/PlantCommunication/XComCfg (IEC, version 4.14.0)
